C01812=1036.838,375.996,367.337,173.070,44.900,158.843
C01813=1036.829,375.750,367.377,173.063,44.896,158.841
C01814=1036.821,375.503,367.418,173.055,44.893,158.839
C01815=1036.813,375.256,367.459,173.047,44.889,158.838
C01816=1036.805,375.010,367.499,173.040,44.886,158.836
C01817=1036.796,374.763,367.540,173.033,44.883,158.835
C01818=1036.787,374.517,367.580,173.026,44.879,158.833
C01819=1036.779,374.270,367.621,173.019,44.876,158.832
C01820=1036.771,374.024,367.662,173.012,44.872,158.830
C01821=1036.763,373.778,367.703,173.005,44.869,158.828
C01822=1036.753,373.531,367.743,172.998,44.865,158.827
C01823=1036.746,373.284,367.783,172.991,44.862,158.825
C01824=1036.738,373.038,367.824,172.984,44.858,158.824
C01825=1036.729,372.791,367.865,172.976,44.855,158.822
C01826=1036.721,372.545,367.905,172.969,44.851,158.821
C01827=1036.712,372.298,367.944,172.962,44.848,158.819
C01828=1036.704,372.052,367.985,172.955,44.845,158.818
C01829=1036.696,371.805,368.026,172.948,44.841,158.816
C01830=1036.688,371.558,368.067,172.941,44.838,158.815
C01831=1036.679,371.312,368.106,172.934,44.835,158.813
C01832=1036.671,371.066,368.147,172.927,44.832,158.812
C01833=1036.664,370.819,368.187,172.921,44.828,158.810
C01834=1036.655,370.572,368.228,172.914,44.825,158.809
C01835=1036.647,370.325,368.267,172.907,44.821,158.807
C01836=1036.639,370.079,368.308,172.900,44.818,158.806
C01837=1036.631,369.832,368.348,172.893,44.814,158.804
C01838=1036.622,369.586,368.388,172.886,44.811,158.803
C01839=1036.614,369.339,368.427,172.879,44.808,158.801
C01840=1036.605,369.092,368.467,172.872,44.805,158.800
C01841=1036.596,368.846,368.507,172.865,44.802,158.798
C01842=1036.589,368.599,368.547,172.859,44.799,158.797
C01843=1036.580,368.352,368.586,172.852,44.796,158.795
C01844=1036.573,368.105,368.626,172.845,44.792,158.794
C01845=1036.564,367.859,368.666,172.838,44.789,158.792
C01846=1036.556,367.612,368.706,172.831,44.786,158.791
C01847=1036.548,367.366,368.746,172.825,44.783,158.790
C01848=1036.539,367.119,368.785,172.818,44.780,158.788
C01849=1036.531,366.872,368.825,172.811,44.777,158.787
C01850=1036.523,366.626,368.864,172.805,44.774,158.785
C01851=1036.515,366.379,368.904,172.798,44.771,158.784
C01852=1036.507,366.132,368.943,172.791,44.768,158.782
C01853=1036.499,365.885,368.983,172.785,44.764,158.781
C01854=1036.491,365.639,369.023,172.778,44.761,158.780
C01855=1036.482,365.392,369.062,172.771,44.758,158.778
C01856=1036.474,365.145,369.102,172.765,44.755,158.777
C01857=1036.466,364.899,369.141,172.758,44.752,158.775
C01858=1036.459,364.651,369.180,172.752,44.749,158.774
C01859=1036.450,364.404,369.220,172.745,44.746,158.773
C01860=1036.438,364.022,369.281,172.734,44.741,158.770
C01861=1036.426,363.640,369.342,172.725,44.737,158.768
C01862=1036.413,363.258,369.402,172.715,44.732,158.766
C01863=1036.401,362.876,369.463,172.704,44.728,158.764
C01864=1036.393,362.629,369.503,172.698,44.724,158.763
C01865=1036.385,362.382,369.542,172.692,44.721,158.761
C01866=1036.377,362.136,369.581,172.685,44.719,158.760
C01867=1036.369,361.889,369.621,172.679,44.716,158.759
C01868=1036.361,361.642,369.659,172.672,44.712,158.757
C01869=1036.353,361.395,369.699,172.666,44.710,158.756
C01870=1036.345,361.148,369.737,172.659,44.707,158.755
C01871=1036.338,360.901,369.776,172.653,44.704,158.754
C01872=1036.329,360.654,369.815,172.647,44.701,158.752
C01873=1036.321,360.407,369.854,172.640,44.699,158.751
C01874=1036.313,360.161,369.893,172.634,44.695,158.750
C01875=1036.305,359.914,369.931,172.628,44.693,158.748
C01876=1036.297,359.667,369.970,172.621,44.691,158.747
C01877=1036.289,359.420,370.008,172.615,44.687,158.746
C01878=1036.281,359.174,370.048,172.609,44.685,158.745
C01879=1036.274,358.926,370.087,172.603,44.681,158.743
C01880=1036.266,358.680,370.125,172.596,44.679,158.742
C01881=1036.258,358.432,370.164,172.590,44.676,158.741
C01882=1036.250,358.185,370.202,172.584,44.674,158.740
C01883=1036.242,357.939,370.241,172.577,44.671,158.738
C01884=1036.234,357.691,370.279,172.571,44.668,158.737
C01885=1036.226,357.446,370.318,172.565,44.666,158.736
C01886=1036.218,357.198,370.357,172.559,44.663,158.734
C01887=1036.210,356.952,370.395,172.553,44.660,158.733
C01888=1036.202,356.705,370.434,172.546,44.657,158.732
C01889=1036.195,356.458,370.472,172.541,44.655,158.731
C01890=1036.187,356.211,370.510,172.534,44.652,158.729
C01891=1036.179,355.964,370.548,172.529,44.649,158.728
C01892=1036.171,355.717,370.587,172.522,44.647,158.727
C01893=1036.163,355.469,370.625,172.516,44.644,158.726
C01894=1036.155,355.223,370.663,172.510,44.642,158.725
C01895=1036.147,354.976,370.702,172.504,44.639,158.723
C01896=1036.140,354.728,370.740,172.498,44.636,158.722
C01897=1036.132,354.482,370.777,172.491,44.634,158.721
C01898=1036.124,354.235,370.816,172.486,44.631,158.720
C01899=1036.116,353.989,370.854,172.479,44.629,158.719
C01900=1036.108,353.741,370.892,172.474,44.626,158.717
C01901=1036.101,353.494,370.930,172.467,44.624,158.716
C01902=1036.093,353.246,370.968,172.462,44.621,158.715
C01903=1036.085,353.000,371.006,172.455,44.618,158.714
C01904=1036.077,352.754,371.044,172.450,44.616,158.713
C01905=1036.069,352.506,371.082,172.443,44.614,158.711
C01906=1036.062,352.259,371.120,172.438,44.611,158.710
C01907=1036.054,352.012,371.158,172.432,44.608,158.709
C01908=1036.046,351.765,371.196,172.426,44.606,158.708
C01909=1036.039,351.518,371.234,172.420,44.604,158.707
C01910=1036.031,351.271,371.272,172.414,44.601,158.706
C01911=1036.023,351.024,371.309,172.408,44.598,158.704
C01912=1036.015,350.777,371.348,172.402,44.596,158.703
C01913=1036.008,350.530,371.385,172.396,44.594,158.702
C01914=1036.001,350.283,371.423,172.391,44.591,158.701
C01915=1035.993,350.036,371.461,172.385,44.589,158.700
C01916=1035.981,349.660,371.518,172.376,44.585,158.698
C01917=1035.969,349.284,371.575,172.367,44.581,158.696
C01918=1035.957,348.907,371.632,172.358,44.578,158.695
C01919=1035.946,348.531,371.689,172.350,44.574,158.693
C01920=1035.938,348.284,371.727,172.343,44.572,158.692
C01921=1035.931,348.037,371.765,172.338,44.570,158.691
C01922=1035.923,347.790,371.802,172.333,44.567,158.690
C01923=1035.916,347.543,371.839,172.326,44.565,158.689
C01924=1035.908,347.296,371.876,172.321,44.563,158.688
C01925=1035.900,347.048,371.914,172.315,44.560,158.686
C01926=1035.893,346.801,371.952,172.309,44.558,158.685
C01927=1035.885,346.554,371.989,172.304,44.556,158.684
C01928=1035.877,346.307,372.026,172.298,44.553,158.683
C01929=1035.869,346.060,372.063,172.292,44.551,158.682
C01930=1035.862,345.813,372.101,172.287,44.549,158.681
C01931=1035.854,345.566,372.137,172.281,44.547,158.680
C01932=1035.847,345.319,372.174,172.275,44.545,158.679
C01933=1035.840,345.072,372.212,172.270,44.542,158.678
C01934=1035.832,344.825,372.249,172.264,44.540,158.677
C01935=1035.825,344.578,372.286,172.259,44.538,158.676
C01936=1035.817,344.330,372.323,172.253,44.536,158.675
C01937=1035.810,344.083,372.360,172.247,44.533,158.674
C01938=1035.802,343.836,372.397,172.242,44.531,158.673
C01939=1035.795,343.589,372.434,172.237,44.529,158.672
C01940=1035.787,343.342,372.471,172.230,44.527,158.671
C01941=1035.780,343.094,372.508,172.225,44.525,158.670
C01942=1035.772,342.848,372.545,172.220,44.522,158.668
C01943=1035.764,342.600,372.581,172.214,44.520,158.667
C01944=1035.757,342.353,372.619,172.208,44.518,158.666
C01945=1035.749,342.106,372.655,172.203,44.516,158.665
C01946=1035.742,341.858,372.693,172.197,44.514,158.664
C01947=1035.734,341.611,372.729,172.192,44.512,158.663
C01948=1035.727,341.364,372.766,172.187,44.510,158.662
C01949=1035.719,341.116,372.803,172.181,44.508,158.661
C01950=1035.712,340.870,372.839,172.175,44.506,158.660
C01951=1035.705,340.623,372.876,172.170,44.503,158.659
C01952=1035.697,340.376,372.913,172.165,44.502,158.658
C01953=1035.689,340.128,372.949,172.160,44.500,158.657
C01954=1035.682,339.881,372.985,172.153,44.498,158.656
C01955=1035.674,339.634,373.023,172.148,44.496,158.655
C01956=1035.667,339.386,373.059,172.143,44.493,158.654
C01957=1035.660,339.140,373.095,172.138,44.492,158.653
C01958=1035.652,338.892,373.131,172.133,44.490,158.652
C01959=1035.644,338.645,373.168,172.127,44.488,158.651
C01960=1035.637,338.397,373.205,172.121,44.486,158.650
C01961=1035.629,338.150,373.241,172.116,44.483,158.649
C01962=1035.622,337.903,373.277,172.111,44.482,158.649
C01963=1035.615,337.656,373.313,172.106,44.480,158.647
C01964=1035.608,337.408,373.350,172.100,44.477,158.646
C01965=1035.600,337.161,373.386,172.095,44.476,158.646
C01966=1035.593,336.915,373.423,172.090,44.474,158.645
C01967=1035.585,336.667,373.459,172.085,44.472,158.644
C01968=1035.577,336.420,373.495,172.080,44.470,158.643
C01969=1035.570,336.172,373.532,172.073,44.468,158.642
C01970=1035.563,335.925,373.568,172.068,44.466,158.641
C01971=1035.556,335.678,373.604,172.063,44.464,158.640
C01972=1035.545,335.298,373.660,172.055,44.461,158.638
C01973=1035.533,334.919,373.715,172.048,44.458,158.637
C01974=1035.522,334.538,373.770,172.040,44.455,158.636
C01975=1035.511,334.159,373.825,172.031,44.453,158.634
C01976=1035.503,333.911,373.862,172.026,44.451,158.633
C01977=1035.496,333.665,373.897,172.021,44.449,158.632
C01978=1035.489,333.417,373.933,172.016,44.447,158.631
C01979=1035.481,333.170,373.969,172.010,44.445,158.630
C01980=1035.474,332.922,374.005,172.005,44.444,158.630
C01981=1035.466,332.675,374.041,172.000,44.442,158.629
C01982=1035.459,332.428,374.076,171.995,44.440,158.628
C01983=1035.451,332.180,374.112,171.990,44.438,158.627
C01984=1035.444,331.934,374.148,171.985,44.437,158.626
C01985=1035.437,331.686,374.183,171.980,44.435,158.625
C01986=1035.429,331.439,374.219,171.975,44.433,158.624
C01987=1035.422,331.191,374.255,171.970,44.431,158.623
C01988=1035.415,330.944,374.290,171.964,44.429,158.622
C01989=1035.408,330.696,374.326,171.959,44.428,158.622
C01990=1035.401,330.449,374.362,171.954,44.426,158.621
C01991=1035.393,330.202,374.398,171.949,44.424,158.620
C01992=1035.386,329.955,374.433,171.944,44.423,158.619
C01993=1035.379,329.706,374.469,171.939,44.421,158.618
C01994=1035.372,329.460,374.505,171.934,44.419,158.617
C01995=1035.364,329.212,374.540,171.929,44.418,158.616
C01996=1035.357,328.965,374.576,171.924,44.416,158.616
C01997=1035.350,328.718,374.611,171.919,44.414,158.615
C01998=1035.342,328.470,374.647,171.914,44.412,158.614
C01999=1035.335,328.223,374.682,171.909,44.411,158.613
C02000=1035.328,327.975,374.717,171.904,44.409,158.612
C02001=1035.320,327.728,374.752,171.899,44.407,158.611
C02002=1035.313,327.480,374.787,171.894,44.406,158.610
C02003=1035.305,327.233,374.823,171.890,44.404,158.610
C02004=1035.298,326.986,374.858,171.885,44.403,158.609
C02005=1035.290,326.738,374.893,171.880,44.401,158.608
C02006=1035.284,326.491,374.928,171.875,44.400,158.607
C02007=1035.275,326.243,374.963,171.870,44.398,158.606
C02008=1035.269,325.996,374.998,171.865,44.397,158.606
C02009=1035.261,325.749,375.032,171.860,44.395,158.605
C02010=1035.254,325.501,375.068,171.855,44.394,158.604
C02011=1035.246,325.254,375.102,171.850,44.392,158.603
C02012=1035.240,325.006,375.138,171.845,44.390,158.602
C02013=1035.231,324.758,375.172,171.840,44.389,158.602
C02014=1035.225,324.511,375.208,171.835,44.388,158.601
C02015=1035.217,324.264,375.242,171.830,44.386,158.600
C02016=1035.210,324.016,375.278,171.826,44.384,158.599
C02017=1035.202,323.769,375.312,171.821,44.383,158.598
C02018=1035.196,323.522,375.347,171.816,44.382,158.598
C02019=1035.188,323.275,375.382,171.811,44.380,158.597
C02020=1035.181,323.026,375.417,171.806,44.379,158.596
C02021=1035.173,322.779,375.452,171.801,44.377,158.595
C02022=1035.167,322.531,375.486,171.796,44.376,158.594
C02023=1035.159,322.284,375.521,171.791,44.374,158.594
C02024=1035.152,322.036,375.556,171.787,44.373,158.593
C02025=1035.144,321.789,375.591,171.783,44.372,158.592
C02026=1035.138,321.542,375.626,171.778,44.370,158.591
C02027=1035.130,321.294,375.660,171.773,44.368,158.590
C02028=1035.119,320.910,375.714,171.765,44.366,158.589
C02029=1035.108,320.526,375.768,171.758,44.364,158.588
C02030=1035.096,320.142,375.822,171.750,44.362,158.587
C02031=1035.085,319.757,375.875,171.743,44.360,158.586
C02032=1035.079,319.510,375.910,171.739,44.358,158.585
C02033=1035.071,319.262,375.944,171.734,44.357,158.584
C02034=1035.065,319.015,375.979,171.729,44.356,158.584
C02035=1035.057,318.767,376.013,171.724,44.354,158.583
C02036=1035.051,318.519,376.048,171.720,44.353,158.582
C02037=1035.043,318.272,376.082,171.715,44.351,158.581
C02038=1035.037,318.024,376.117,171.711,44.350,158.581
C02039=1035.029,317.777,376.151,171.706,44.349,158.580
C02040=1035.022,317.530,376.186,171.701,44.347,158.579
C02041=1035.015,317.282,376.220,171.697,44.346,158.578
C02042=1035.008,317.035,376.254,171.692,44.344,158.577
C02043=1035.001,316.787,376.289,171.687,44.343,158.577
C02044=1034.994,316.540,376.323,171.683,44.342,158.576
C02045=1034.987,316.292,376.358,171.678,44.340,158.575
C02046=1034.980,316.045,376.392,171.673,44.339,158.575
C02047=1034.973,315.798,376.427,171.668,44.338,158.574
C02048=1034.966,315.550,376.461,171.665,44.337,158.573
C02049=1034.959,315.302,376.495,171.660,44.335,158.572
C02050=1034.952,315.055,376.530,171.655,44.334,158.572
C02051=1034.945,314.808,376.563,171.651,44.332,158.571
C02052=1034.939,314.560,376.598,171.646,44.331,158.570
C02053=1034.932,314.313,376.632,171.641,44.330,158.570
C02054=1034.924,314.065,376.666,171.637,44.328,158.569
C02055=1034.918,313.817,376.701,171.633,44.327,158.568
C02056=1034.911,313.569,376.734,171.628,44.326,158.567
C02057=1034.904,313.322,376.770,171.624,44.325,158.567
C02058=1034.897,313.075,376.803,171.619,44.324,158.566
C02059=1034.890,312.827,376.837,171.614,44.322,158.565
C02060=1034.884,312.579,376.871,171.610,44.321,158.565
C02061=1034.876,312.331,376.905,171.606,44.320,158.564
C02062=1034.870,312.084,376.940,171.601,44.318,158.563
C02063=1034.863,311.837,376.974,171.597,44.317,158.562
C02064=1034.856,311.589,377.008,171.592,44.316,158.562
C02065=1034.849,311.342,377.041,171.587,44.315,158.561
C02066=1034.841,311.094,377.075,171.584,44.314,158.560
C02067=1034.834,310.846,377.109,171.579,44.313,158.560
C02068=1034.828,310.599,377.142,171.574,44.312,158.559
C02069=1034.820,310.352,377.175,171.570,44.310,158.558
C02070=1034.813,310.104,377.209,171.565,44.309,158.558
C02071=1034.806,309.856,377.243,171.561,44.308,158.557
C02072=1034.798,309.608,377.276,171.557,44.307,158.557
C02073=1034.791,309.361,377.310,171.552,44.306,158.556
C02074=1034.784,309.114,377.342,171.547,44.305,158.555
C02075=1034.777,308.866,377.376,171.544,44.304,158.555
C02076=1034.770,308.618,377.410,171.539,44.303,158.554
C02077=1034.763,308.371,377.444,171.534,44.302,158.553
C02078=1034.756,308.123,377.477,171.530,44.301,158.553
C02079=1034.748,307.876,377.510,171.526,44.300,158.552
C02080=1034.741,307.628,377.544,171.521,44.299,158.551
C02081=1034.734,307.380,377.577,171.517,44.297,158.551
C02082=1034.728,307.133,377.610,171.512,44.296,158.550
C02083=1034.720,306.885,377.643,171.508,44.295,158.549
C02084=1034.710,306.505,377.694,171.502,44.294,158.548
C02085=1034.698,306.126,377.746,171.494,44.292,158.547
C02086=1034.688,305.746,377.797,171.488,44.291,158.547
C02087=1034.677,305.367,377.848,171.481,44.290,158.546
C02088=1034.670,305.120,377.881,171.477,44.288,158.545
C02089=1034.663,304.872,377.914,171.473,44.287,158.544
C02090=1034.656,304.624,377.947,171.469,44.286,158.544
C02091=1034.649,304.377,377.980,171.464,44.285,158.543
C02092=1034.642,304.129,378.013,171.460,44.284,158.542
C02093=1034.636,303.881,378.046,171.456,44.283,158.542
C02094=1034.628,303.634,378.079,171.451,44.282,158.541
C02095=1034.621,303.386,378.113,171.447,44.281,158.541
C02096=1034.614,303.139,378.146,171.443,44.280,158.540
C02097=1034.607,302.890,378.179,171.439,44.280,158.539
C02098=1034.601,302.643,378.213,171.434,44.279,158.539
C02099=1034.593,302.395,378.245,171.431,44.277,158.538
C02100=1034.587,302.148,378.278,171.426,44.276,158.538
C02101=1034.580,301.900,378.312,171.422,44.276,158.537
C02102=1034.573,301.653,378.344,171.418,44.275,158.536
C02103=1034.566,301.405,378.377,171.414,44.273,158.536
C02104=1034.559,301.158,378.410,171.409,44.272,158.535
C02105=1034.552,300.909,378.443,171.406,44.272,158.535
C02106=1034.546,300.662,378.476,171.401,44.271,158.534
C02107=1034.538,300.414,378.509,171.397,44.270,158.533
C02108=1034.532,300.167,378.542,171.393,44.269,158.533
C02109=1034.525,299.919,378.575,171.389,44.268,158.532
C02110=1034.519,299.671,378.608,171.384,44.267,158.532
C02111=1034.511,299.423,378.641,171.380,44.266,158.531
C02112=1034.505,299.175,378.673,171.376,44.265,158.530
C02113=1034.498,298.928,378.706,171.372,44.264,158.530
C02114=1034.490,298.680,378.739,171.367,44.264,158.529
C02115=1034.484,298.433,378.772,171.364,44.262,158.529
C02116=1034.477,298.184,378.805,171.359,44.261,158.528
C02117=1034.471,297.937,378.838,171.355,44.261,158.528
C02118=1034.464,297.690,378.870,171.352,44.260,158.527
C02119=1034.457,297.441,378.903,171.347,44.259,158.526
C02120=1034.451,297.194,378.936,171.343,44.258,158.526
C02121=1034.444,296.946,378.969,171.339,44.257,158.525
C02122=1034.437,296.698,379.001,171.335,44.256,158.525
C02123=1034.431,296.451,379.034,171.330,44.255,158.524
C02124=1034.424,296.203,379.067,171.327,44.255,158.524
C02125=1034.417,295.955,379.099,171.323,44.253,158.523
C02126=1034.410,295.707,379.132,171.318,44.252,158.522
C02127=1034.404,295.460,379.165,171.315,44.252,158.522
C02128=1034.397,295.211,379.198,171.310,44.251,158.521
C02129=1034.390,294.964,379.230,171.307,44.250,158.521
C02130=1034.384,294.717,379.263,171.303,44.249,158.520
C02131=1034.376,294.469,379.295,171.298,44.248,158.520
C02132=1034.370,294.221,379.328,171.295,44.248,158.519
C02133=1034.363,293.973,379.359,171.290,44.247,158.518
C02134=1034.356,293.726,379.391,171.286,44.246,158.518
C02135=1034.349,293.478,379.425,171.283,44.246,158.518
C02136=1034.343,293.230,379.456,171.278,44.245,158.517
C02137=1034.336,292.982,379.489,171.275,44.244,158.516
C02138=1034.329,292.734,379.521,171.270,44.243,158.516
C02139=1034.322,292.487,379.553,171.266,44.242,158.515
C02140=1034.312,292.124,379.600,171.261,44.241,158.515
C02141=1034.301,291.761,379.647,171.255,44.241,158.514
C02142=1034.292,291.399,379.694,171.249,44.239,158.513
C02143=1034.282,291.036,379.741,171.243,44.238,158.512
C02144=1034.275,290.789,379.773,171.240,44.238,158.512
C02145=1034.268,290.540,379.805,171.235,44.237,158.511
C02146=1034.261,290.293,379.837,171.231,44.236,158.511
C02147=1034.254,290.045,379.870,171.228,44.235,158.510
C02148=1034.248,289.797,379.902,171.223,44.235,158.510
C02149=1034.241,289.549,379.933,171.220,44.234,158.509
C02150=1034.234,289.301,379.966,171.216,44.233,158.509
C02151=1034.227,289.053,379.997,171.212,44.233,158.508
C02152=1034.220,288.806,380.029,171.208,44.232,158.508
C02153=1034.214,288.558,380.061,171.205,44.231,158.507
C02154=1034.207,288.311,380.093,171.200,44.231,158.507
C02155=1034.200,288.063,380.125,171.196,44.230,158.506
C02156=1034.193,287.814,380.157,171.193,44.229,158.506
C02157=1034.186,287.567,380.189,171.188,44.229,158.505
C02158=1034.180,287.319,380.221,171.185,44.228,158.505
C02159=1034.173,287.071,380.252,171.181,44.228,158.504
C02160=1034.166,286.823,380.284,171.177,44.227,158.504
C02161=1034.159,286.576,380.316,171.173,44.226,158.503
C02162=1034.153,286.328,380.347,171.170,44.226,158.503
C02163=1034.145,286.079,380.379,171.165,44.225,158.502
C02164=1034.138,285.832,380.411,171.162,44.225,158.502
C02165=1034.132,285.584,380.443,171.158,44.224,158.501
C02166=1034.125,285.336,380.474,171.154,44.224,158.501
C02167=1034.118,285.088,380.505,171.150,44.223,158.500
C02168=1034.111,284.840,380.537,171.147,44.223,158.500
C02169=1034.105,284.592,380.568,171.142,44.222,158.500
C02170=1034.098,284.344,380.600,171.139,44.221,158.499
C02171=1034.091,284.096,380.631,171.135,44.221,158.499
C02172=1034.084,283.848,380.663,171.131,44.220,158.498
C02173=1034.077,283.601,380.695,171.127,44.220,158.498
C02174=1034.070,283.353,380.726,171.123,44.219,158.497
C02175=1034.063,283.105,380.758,171.120,44.219,158.497
C02176=1034.057,282.857,380.789,171.115,44.218,158.496
C02177=1034.049,282.609,380.820,171.112,44.217,158.496
C02178=1034.043,282.361,380.852,171.108,44.217,158.495
C02179=1034.036,282.113,380.883,171.104,44.216,158.495
C02180=1034.029,281.866,380.914,171.100,44.216,158.494
C02181=1034.022,281.618,380.946,171.097,44.215,158.494
C02182=1034.016,281.369,380.977,171.093,44.215,158.493
C02183=1034.009,281.121,381.008,171.089,44.215,158.493
C02184=1034.002,280.873,381.039,171.086,44.214,158.493
C02185=1033.996,280.625,381.071,171.082,44.213,158.492
C02186=1033.989,280.378,381.102,171.079,44.213,158.492
C02187=1033.982,280.130,381.134,171.075,44.212,158.491
C02188=1033.976,279.882,381.165,171.071,44.212,158.491
C02189=1033.969,279.634,381.197,171.067,44.211,158.490
C02190=1033.962,279.386,381.228,171.064,44.211,158.490
C02191=1033.956,279.138,381.258,171.060,44.211,158.490
C02192=1033.950,278.890,381.290,171.056,44.210,158.489
C02193=1033.943,278.642,381.321,171.052,44.209,158.489
C02194=1033.935,278.395,381.352,171.049,44.209,158.488
C02195=1033.929,278.147,381.384,171.045,44.208,158.488
C02196=1033.920,277.796,381.427,171.040,44.208,158.487
C02197=1033.910,277.445,381.471,171.035,44.207,158.486
C02198=1033.900,277.095,381.515,171.029,44.207,158.486
C02199=1033.891,276.744,381.559,171.025,44.206,158.485
C02200=1033.883,276.497,381.590,171.020,44.206,158.485
C02201=1033.877,276.248,381.620,171.017,44.205,158.484
C02202=1033.870,276.000,381.652,171.013,44.205,158.484
C02203=1033.864,275.752,381.682,171.010,44.205,158.484
C02204=1033.856,275.504,381.713,171.007,44.204,158.483
C02205=1033.850,275.256,381.744,171.002,44.204,158.483
C02206=1033.844,275.009,381.775,170.999,44.204,158.482
C02207=1033.836,274.761,381.806,170.995,44.203,158.482
C02208=1033.830,274.513,381.837,170.992,44.202,158.482
C02209=1033.823,274.265,381.868,170.988,44.202,158.481
C02210=1033.816,274.016,381.898,170.985,44.202,158.481
C02211=1033.809,273.768,381.930,170.980,44.201,158.480
C02212=1033.804,273.521,381.960,170.977,44.201,158.480
C02213=1033.796,273.272,381.990,170.974,44.201,158.480
C02214=1033.790,273.025,382.021,170.970,44.200,158.479
C02215=1033.782,272.776,382.052,170.967,44.200,158.479
C02216=1033.776,272.528,382.083,170.963,44.199,158.478
C02217=1033.770,272.281,382.113,170.959,44.199,158.478
C02218=1033.763,272.032,382.144,170.956,44.199,158.478
C02219=1033.756,271.784,382.175,170.952,44.199,158.477
C02220=1033.749,271.536,382.205,170.949,44.198,158.477
C02221=1033.742,271.288,382.236,170.945,44.198,158.476
C02222=1033.736,271.041,382.266,170.942,44.197,158.476
C02223=1033.729,270.792,382.297,170.939,44.197,158.476
C02224=1033.722,270.544,382.327,170.934,44.197,158.475
C02225=1033.716,270.296,382.358,170.931,44.196,158.475
C02226=1033.709,270.049,382.388,170.927,44.196,158.474
C02227=1033.702,269.800,382.419,170.924,44.196,158.474
C02228=1033.695,269.552,382.449,170.921,44.196,158.474
C02229=1033.689,269.303,382.480,170.917,44.195,158.473
C02230=1033.682,269.056,382.510,170.914,44.195,158.473
C02231=1033.675,268.808,382.541,170.910,44.194,158.472
C02232=1033.668,268.560,382.571,170.906,44.195,158.472
C02233=1033.662,268.312,382.601,170.903,44.194,158.472
C02234=1033.655,268.064,382.632,170.899,44.194,158.471
C02235=1033.648,267.816,382.662,170.896,44.194,158.471
C02236=1033.642,267.567,382.692,170.893,44.193,158.471
C02237=1033.635,267.320,382.722,170.889,44.193,158.470
C02238=1033.628,267.071,382.752,170.886,44.193,158.470
C02239=1033.622,266.823,382.783,170.883,44.193,158.470
C02240=1033.615,266.575,382.813,170.879,44.192,158.469
C02241=1033.608,266.327,382.843,170.876,44.192,158.469
C02242=1033.602,266.079,382.874,170.871,44.192,158.468
C02243=1033.595,265.831,382.903,170.868,44.192,158.468
C02244=1033.588,265.583,382.934,170.865,44.192,158.468
C02245=1033.581,265.335,382.964,170.861,44.192,158.467
C02246=1033.575,265.087,382.994,170.858,44.191,158.467
C02247=1033.568,264.839,383.024,170.855,44.191,158.467
C02248=1033.561,264.591,383.054,170.851,44.191,158.466
C02249=1033.555,264.343,383.085,170.848,44.190,158.466
C02250=1033.548,264.094,383.115,170.845,44.190,158.466
C02251=1033.541,263.847,383.144,170.841,44.190,158.465
C02252=1033.532,263.501,383.186,170.836,44.190,158.465
C02253=1033.522,263.155,383.227,170.831,44.190,158.464
C02254=1033.513,262.808,383.270,170.827,44.189,158.464
C02255=1033.504,262.463,383.312,170.822,44.189,158.463
C02256=1033.497,262.215,383.341,170.819,44.189,158.463
C02257=1033.490,261.966,383.371,170.816,44.189,158.463
C02258=1033.484,261.719,383.402,170.812,44.189,158.462
C02259=1033.477,261.470,383.432,170.809,44.188,158.462
C02260=1033.471,261.222,383.461,170.806,44.188,158.462
C02261=1033.464,260.974,383.491,170.801,44.188,158.461
C02262=1033.457,260.726,383.521,170.798,44.188,158.461
C02263=1033.450,260.478,383.549,170.795,44.188,158.461
C02264=1033.442,260.230,383.580,170.792,44.188,158.460
C02265=1033.436,259.982,383.609,170.788,44.188,158.460
C02266=1033.429,259.734,383.639,170.785,44.187,158.460
C02267=1033.422,259.486,383.669,170.781,44.187,158.459
C02268=1033.416,259.237,383.698,170.778,44.187,158.459
C02269=1033.408,258.989,383.728,170.775,44.187,158.459
C02270=1033.401,258.741,383.757,170.772,44.187,158.458
C02271=1033.394,258.493,383.787,170.768,44.187,158.458
C02272=1033.388,258.245,383.816,170.765,44.187,158.458
C02273=1033.381,257.997,383.846,170.762,44.187,158.458
C02274=1033.375,257.748,383.875,170.759,44.187,158.457
C02275=1033.368,257.500,383.904,170.755,44.187,158.457
C02276=1033.361,257.252,383.934,170.752,44.187,158.457
C02277=1033.354,257.004,383.963,170.749,44.187,158.456
C02278=1033.347,256.756,383.993,170.745,44.187,158.456
C02279=1033.340,256.507,384.022,170.742,44.187,158.456
C02280=1033.334,256.260,384.052,170.739,44.187,158.455
C02281=1033.327,256.011,384.081,170.735,44.187,158.455
C02282=1033.321,255.763,384.110,170.732,44.187,158.455
C02283=1033.313,255.515,384.140,170.729,44.186,158.454
C02284=1033.306,255.267,384.169,170.726,44.186,158.454
C02285=1033.300,255.018,384.198,170.722,44.186,158.454
C02286=1033.293,254.770,384.228,170.719,44.186,158.453
C02287=1033.286,254.522,384.257,170.716,44.186,158.453
C02288=1033.280,254.273,384.286,170.713,44.186,158.453
C02289=1033.273,254.026,384.316,170.709,44.186,158.453
C02290=1033.266,253.777,384.345,170.706,44.186,158.452
C02291=1033.260,253.529,384.374,170.703,44.186,158.452
C02292=1033.253,253.280,384.403,170.699,44.186,158.452
C02293=1033.246,253.033,384.433,170.696,44.186,158.451
C02294=1033.240,252.785,384.462,170.693,44.186,158.451
C02295=1033.233,252.536,384.492,170.690,44.186,158.451
C02296=1033.226,252.288,384.520,170.686,44.186,158.450
C02297=1033.219,252.040,384.550,170.683,44.186,158.450
C02298=1033.213,251.792,384.579,170.680,44.186,158.450
C02299=1033.206,251.544,384.608,170.677,44.186,158.450
C02300=1033.200,251.295,384.638,170.673,44.186,158.449
C02301=1033.193,251.047,384.667,170.670,44.186,158.449
C02302=1033.186,250.799,384.695,170.668,44.186,158.449
C02303=1033.179,250.551,384.725,170.664,44.186,158.448
C02304=1033.173,250.303,384.754,170.661,44.186,158.448
C02305=1033.167,250.054,384.783,170.658,44.186,158.448
C02306=1033.160,249.806,384.813,170.655,44.186,158.448
C02307=1033.153,249.558,384.841,170.651,44.186,158.447
C02308=1033.144,249.210,384.883,170.647,44.186,158.447
C02309=1033.135,248.863,384.923,170.643,44.186,158.447
C02310=1033.126,248.515,384.964,170.638,44.186,158.446
C02311=1033.117,248.169,385.004,170.634,44.186,158.446
C02312=1033.109,247.920,385.033,170.631,44.186,158.445
C02313=1033.103,247.672,385.062,170.627,44.186,158.445
C02314=1033.097,247.424,385.091,170.624,44.186,158.445
C02315=1033.091,247.176,385.120,170.621,44.186,158.445
C02316=1033.084,246.927,385.149,170.618,44.186,158.444
C02317=1033.077,246.679,385.178,170.616,44.186,158.444
C02318=1033.070,246.431,385.207,170.612,44.186,158.444
C02319=1033.064,246.183,385.236,170.609,44.186,158.444
C02320=1033.058,245.935,385.265,170.606,44.186,158.443
C02321=1033.051,245.686,385.294,170.603,44.186,158.443
C02322=1033.044,245.438,385.323,170.599,44.186,158.443
C02323=1033.038,245.190,385.352,170.596,44.186,158.442
C02324=1033.032,244.942,385.381,170.594,44.186,158.442
C02325=1033.025,244.694,385.410,170.590,44.186,158.442
C02326=1033.018,244.445,385.439,170.587,44.186,158.441
C02327=1033.012,244.196,385.467,170.584,44.186,158.441
C02328=1033.006,243.948,385.496,170.581,44.186,158.441
C02329=1032.999,243.700,385.525,170.578,44.186,158.441
C02330=1032.992,243.452,385.554,170.574,44.186,158.440
C02331=1032.985,243.203,385.582,170.572,44.186,158.440
C02332=1032.979,242.955,385.611,170.569,44.187,158.440
C02333=1032.972,242.707,385.639,170.566,44.187,158.440
C02334=1032.966,242.459,385.668,170.563,44.187,158.439
C02335=1032.959,242.211,385.696,170.559,44.187,158.439
C02336=1032.952,241.962,385.725,170.556,44.187,158.439
C02337=1032.945,241.714,385.754,170.554,44.187,158.439
C02338=1032.939,241.465,385.782,170.551,44.187,158.438
C02339=1032.932,241.217,385.811,170.547,44.187,158.438
C02340=1032.926,240.969,385.840,170.544,44.187,158.438
C02341=1032.919,240.721,385.867,170.541,44.188,158.438
C02342=1032.913,240.473,385.896,170.538,44.188,158.437
C02343=1032.906,240.223,385.925,170.536,44.187,158.437
C02344=1032.899,239.975,385.954,170.533,44.188,158.437
C02345=1032.892,239.728,385.982,170.529,44.188,158.437
C02346=1032.886,239.479,386.010,170.526,44.188,158.436
C02347=1032.879,239.231,386.038,170.523,44.188,158.436
C02348=1032.873,238.983,386.067,170.520,44.188,158.436
C02349=1032.866,238.735,386.095,170.517,44.188,158.436
C02350=1032.859,238.486,386.123,170.514,44.189,158.436
C02351=1032.852,238.237,386.151,170.511,44.189,158.435
C02352=1032.846,237.989,386.180,170.508,44.189,158.435
C02353=1032.839,237.741,386.208,170.505,44.189,158.435
C02354=1032.832,237.493,386.236,170.502,44.189,158.435
C02355=1032.826,237.244,386.264,170.499,44.190,158.434
C02356=1032.819,236.996,386.293,170.496,44.190,158.434
C02357=1032.812,236.748,386.321,170.493,44.190,158.434
C02358=1032.806,236.499,386.348,170.490,44.190,158.434
C02359=1032.798,236.251,386.377,170.487,44.190,158.433
C02360=1032.792,236.002,386.405,170.485,44.191,158.433
C02361=1032.785,235.754,386.433,170.481,44.191,158.433
C02362=1032.778,235.506,386.462,170.478,44.191,158.433
C02363=1032.772,235.257,386.489,170.475,44.191,158.433
C02364=1032.762,234.904,386.529,170.471,44.191,158.432
C02365=1032.753,234.551,386.570,170.466,44.192,158.432
C02366=1032.743,234.198,386.609,170.462,44.192,158.432
C02367=1032.734,233.845,386.649,170.458,44.193,158.431
C02368=1032.727,233.596,386.677,170.456,44.192,158.431
C02369=1032.721,233.348,386.706,170.453,44.193,158.431
C02370=1032.714,233.099,386.733,170.450,44.193,158.431
C02371=1032.707,232.851,386.762,170.446,44.193,158.430
C02372=1032.701,232.603,386.789,170.444,44.193,158.430
C02373=1032.694,232.354,386.817,170.441,44.193,158.430
C02374=1032.688,232.106,386.845,170.438,44.194,158.430
C02375=1032.681,231.857,386.873,170.435,44.194,158.429
C02376=1032.675,231.610,386.901,170.433,44.194,158.429
C02377=1032.668,231.362,386.929,170.429,44.194,158.429
C02378=1032.662,231.113,386.957,170.426,44.195,158.429
C02379=1032.655,230.865,386.984,170.423,44.195,158.429
C02380=1032.648,230.616,387.012,170.421,44.195,158.429
C02381=1032.641,230.368,387.040,170.418,44.195,158.428
C02382=1032.635,230.119,387.068,170.415,44.196,158.428
C02383=1032.628,229.871,387.095,170.411,44.196,158.428
C02384=1032.621,229.623,387.123,170.409,44.196,158.428
C02385=1032.615,229.374,387.151,170.406,44.196,158.427
C02386=1032.608,229.126,387.179,170.403,44.197,158.427
C02387=1032.601,228.878,387.207,170.400,44.197,158.427
C02388=1032.595,228.629,387.235,170.398,44.197,158.427
C02389=1032.588,228.381,387.263,170.395,44.197,158.427
C02390=1032.582,228.132,387.291,170.392,44.198,158.426
C02391=1032.575,227.884,387.319,170.388,44.198,158.426
C02392=1032.568,227.636,387.346,170.386,44.198,158.426
C02393=1032.561,227.387,387.373,170.383,44.199,158.426
C02394=1032.555,227.138,387.400,170.380,44.199,158.426
C02395=1032.548,226.890,387.428,170.378,44.199,158.425
C02396=1032.542,226.642,387.456,170.375,44.200,158.425
C02397=1032.534,226.394,387.483,170.372,44.200,158.425
C02398=1032.528,226.145,387.510,170.369,44.200,158.425
C02399=1032.521,225.897,387.538,170.367,44.201,158.425
C02400=1032.515,225.648,387.565,170.363,44.201,158.424
C02401=1032.508,225.399,387.593,170.360,44.201,158.424
C02402=1032.501,225.151,387.620,170.357,44.202,158.424
C02403=1032.494,224.903,387.648,170.355,44.202,158.424
C02404=1032.487,224.654,387.675,170.352,44.202,158.424
C02405=1032.481,224.406,387.703,170.349,44.203,158.424
C02406=1032.475,224.158,387.730,170.347,44.203,158.423
C02407=1032.467,223.910,387.757,170.344,44.203,158.423
C02408=1032.461,223.661,387.785,170.341,44.204,158.423
C02409=1032.454,223.413,387.812,170.338,44.204,158.423
C02410=1032.448,223.164,387.839,170.335,44.204,158.423
C02411=1032.441,222.915,387.867,170.332,44.205,158.423
C02412=1032.434,222.667,387.894,170.329,44.205,158.422
C02413=1032.427,222.419,387.922,170.327,44.205,158.422
C02414=1032.421,222.170,387.949,170.324,44.206,158.422
C02415=1032.414,221.922,387.976,170.321,44.206,158.422
C02416=1032.407,221.674,388.004,170.319,44.206,158.422
C02417=1032.401,221.425,388.031,170.316,44.207,158.421
C02418=1032.395,221.177,388.058,170.312,44.207,158.421
C02419=1032.388,220.928,388.086,170.310,44.207,158.421
C02420=1032.378,220.568,388.125,170.306,44.208,158.421
C02421=1032.369,220.207,388.165,170.302,44.208,158.421
C02422=1032.359,219.846,388.204,170.298,44.209,158.420
C02423=1032.349,219.485,388.243,170.294,44.209,158.420
C02424=1032.343,219.237,388.271,170.292,44.210,158.420
C02425=1032.336,218.988,388.297,170.288,44.210,158.420
C02426=1032.329,218.740,388.325,170.285,44.211,158.420
C02427=1032.322,218.492,388.351,170.283,44.211,158.419
C02428=1032.316,218.243,388.379,170.280,44.211,158.419
C02429=1032.309,217.994,388.405,170.277,44.212,158.419
C02430=1032.302,217.746,388.433,170.275,44.212,158.419
C02431=1032.295,217.497,388.460,170.272,44.213,158.419
C02432=1032.289,217.249,388.487,170.269,44.213,158.419
C02433=1032.282,217.001,388.513,170.267,44.213,158.418
C02434=1032.275,216.752,388.541,170.264,44.214,158.418
C02435=1032.268,216.503,388.567,170.261,44.214,158.418
C02436=1032.262,216.255,388.594,170.259,44.215,158.418
C02437=1032.255,216.007,388.621,170.256,44.215,158.418
C02438=1032.248,215.758,388.648,170.253,44.215,158.418
C02439=1032.241,215.510,388.675,170.250,44.216,158.418
C02440=1032.235,215.261,388.702,170.247,44.216,158.417
C02441=1032.228,215.013,388.728,170.245,44.217,158.417
C02442=1032.221,214.764,388.756,170.242,44.217,158.417
C02443=1032.215,214.516,388.782,170.239,44.218,158.417
C02444=1032.208,214.267,388.809,170.237,44.218,158.417
C02445=1032.201,214.019,388.836,170.234,44.218,158.417
C02446=1032.195,213.771,388.863,170.232,44.219,158.416
C02447=1032.188,213.522,388.889,170.229,44.219,158.416
C02448=1032.181,213.273,388.917,170.226,44.220,158.416
C02449=1032.175,213.025,388.943,170.223,44.220,158.416
C02450=1032.169,212.776,388.970,170.220,44.220,158.416
C02451=1032.161,212.528,388.997,170.218,44.221,158.416
C02452=1032.155,212.280,389.024,170.215,44.221,158.416
C02453=1032.148,212.031,389.050,170.212,44.222,158.415
C02454=1032.142,211.782,389.077,170.210,44.222,158.415
C02455=1032.135,211.535,389.104,170.207,44.223,158.415
C02456=1032.129,211.286,389.131,170.205,44.223,158.415
C02457=1032.122,211.037,389.158,170.202,44.223,158.415
C02458=1032.115,210.789,389.184,170.199,44.224,158.415
C02459=1032.109,210.540,389.211,170.197,44.224,158.415
C02460=1032.102,210.291,389.237,170.194,44.225,158.414
C02461=1032.095,210.044,389.264,170.192,44.225,158.414
C02462=1032.088,209.794,389.291,170.189,44.226,158.414
C02463=1032.082,209.546,389.317,170.187,44.226,158.414
C02464=1032.075,209.298,389.343,170.184,44.227,158.414
C02465=1032.068,209.049,389.370,170.181,44.228,158.414
C02466=1032.062,208.801,389.396,170.178,44.227,158.413
C02467=1032.055,208.552,389.423,170.175,44.228,158.413
C02468=1032.048,208.303,389.449,170.173,44.228,158.413
C02469=1032.041,208.055,389.475,170.170,44.229,158.413
C02470=1032.035,207.806,389.502,170.167,44.230,158.413
C02471=1032.028,207.558,389.528,170.165,44.230,158.413
C02472=1032.021,207.310,389.556,170.162,44.231,158.413
C02473=1032.014,207.061,389.582,170.160,44.231,158.413
C02474=1032.008,206.813,389.609,170.157,44.232,158.412
C02475=1032.001,206.564,389.635,170.155,44.232,158.412
C02476=1031.991,206.209,389.672,170.151,44.233,158.412
C02477=1031.981,205.854,389.710,170.147,44.234,158.412
C02478=1031.972,205.500,389.747,170.144,44.234,158.412
C02479=1031.963,205.144,389.785,170.140,44.235,158.412
C02480=1031.937,204.095,389.890,169.795,44.131,158.359
C02481=1031.930,203.847,389.915,169.792,44.133,158.359
C02482=1031.924,203.597,389.940,169.789,44.134,158.359
C02483=1031.918,203.349,389.965,169.785,44.135,158.359
C02484=1031.912,203.101,389.990,169.781,44.136,158.359
C02485=1031.906,202.852,390.014,169.777,44.137,158.359
C02486=1031.900,202.603,390.040,169.774,44.139,158.359
C02487=1031.894,202.354,390.064,169.770,44.140,158.359
C02488=1031.889,202.106,390.089,169.767,44.142,158.359
C02489=1031.882,201.857,390.114,169.764,44.143,158.359
C02490=1031.876,201.608,390.139,169.760,44.144,158.358
C02491=1031.870,201.360,390.164,169.756,44.145,158.358
C02492=1031.864,201.111,390.188,169.753,44.146,158.358
C02493=1031.858,200.862,390.214,169.749,44.148,158.358
C02494=1031.852,200.613,390.238,169.745,44.149,158.358
C02495=1031.846,200.365,390.263,169.742,44.151,158.358
C02496=1031.840,200.116,390.287,169.739,44.152,158.358
C02497=1031.833,199.867,390.312,169.735,44.153,158.358
C02498=1031.827,199.618,390.337,169.731,44.155,158.358
C02499=1031.821,199.370,390.360,169.728,44.156,158.358
C02500=1031.815,199.121,390.386,169.725,44.157,158.358
C02501=1031.808,198.872,390.410,169.721,44.159,158.358
C02502=1031.802,198.623,390.434,169.717,44.160,158.358
C02503=1031.796,198.375,390.459,169.714,44.162,158.358
C02504=1031.790,198.126,390.483,169.711,44.164,158.358
C02505=1031.783,197.877,390.507,169.707,44.165,158.358
C02506=1031.778,197.629,390.532,169.704,44.166,158.358
C02507=1031.771,197.380,390.556,169.700,44.168,158.358
C02508=1031.765,197.131,390.581,169.696,44.169,158.358
C02509=1031.759,196.882,390.605,169.693,44.170,158.358
C02510=1031.753,196.634,390.630,169.690,44.172,158.358
C02511=1031.746,196.385,390.654,169.686,44.173,158.358
C02512=1031.741,196.136,390.678,169.683,44.175,158.358
C02513=1031.734,195.887,390.702,169.679,44.177,158.358
C02514=1031.729,195.639,390.727,169.676,44.178,158.358
C02515=1031.722,195.390,390.751,169.673,44.179,158.358
C02516=1031.716,195.141,390.776,169.669,44.181,158.358
C02517=1031.710,194.893,390.800,169.665,44.182,158.358
C02518=1031.704,194.643,390.824,169.662,44.183,158.358
C02519=1031.698,194.395,390.848,169.658,44.185,158.358
C02520=1031.692,194.146,390.872,169.655,44.187,158.358
C02521=1031.685,193.898,390.897,169.652,44.188,158.358
C02522=1031.680,193.649,390.921,169.648,44.190,158.358
C02523=1031.674,193.400,390.945,169.645,44.191,158.358
C02524=1031.668,193.151,390.970,169.642,44.192,158.358
C02525=1031.662,192.902,390.994,169.638,44.194,158.358
C02526=1031.656,192.654,391.018,169.635,44.195,158.358
C02527=1031.650,192.405,391.042,169.631,44.197,158.358
C02528=1031.644,192.156,391.066,169.628,44.199,158.358
C02529=1031.638,191.907,391.090,169.625,44.200,158.358
C02530=1031.632,191.659,391.115,169.621,44.201,158.358
C02531=1031.626,191.410,391.139,169.618,44.203,158.358
C02532=1031.620,191.161,391.162,169.615,44.205,158.358
C02533=1031.614,190.912,391.187,169.612,44.206,158.358
C02534=1031.608,190.664,391.211,169.608,44.207,158.358
C02535=1031.602,190.415,391.235,169.604,44.209,158.358
C02536=1031.596,190.166,391.259,169.601,44.210,158.358
C02537=1031.590,189.917,391.283,169.597,44.211,158.358
C02538=1031.584,189.669,391.307,169.595,44.213,158.358
C02539=1031.578,189.419,391.332,169.591,44.215,158.358
C02540=1031.572,189.171,391.355,169.588,44.216,158.358
C02541=1031.565,188.888,391.383,169.584,44.218,158.358
C02542=1031.558,188.604,391.411,169.581,44.220,158.358
C02543=1031.552,188.320,391.438,169.576,44.221,158.358
C02544=1031.545,188.037,391.465,169.572,44.223,158.358
C02545=1031.539,187.788,391.490,169.570,44.225,158.358
C02546=1031.533,187.539,391.513,169.566,44.226,158.358
C02547=1031.527,187.291,391.537,169.563,44.227,158.358
C02548=1031.521,187.041,391.561,169.559,44.229,158.358
C02549=1031.516,186.792,391.585,169.557,44.231,158.358
C02550=1031.509,186.543,391.609,169.553,44.232,158.358
C02551=1031.504,186.295,391.633,169.550,44.233,158.358
C02552=1031.498,186.047,391.657,169.546,44.235,158.358
C02553=1031.491,185.797,391.680,169.544,44.237,158.358
C02554=1031.486,185.548,391.705,169.540,44.238,158.358
C02555=1031.480,185.300,391.728,169.537,44.239,158.358
C02556=1031.474,185.051,391.753,169.533,44.241,158.358
C02557=1031.468,184.803,391.776,169.531,44.243,158.358
C02558=1031.463,184.553,391.800,169.527,44.244,158.358
C02559=1031.456,184.304,391.824,169.524,44.245,158.358
C02560=1031.450,184.056,391.848,169.520,44.247,158.358
C02561=1031.445,183.808,391.872,169.517,44.249,158.358
C02562=1031.439,183.558,391.895,169.515,44.250,158.358
C02563=1031.433,183.309,391.920,169.511,44.251,158.358
C02564=1031.427,183.061,391.943,169.508,44.253,158.358
C02565=1031.421,182.811,391.967,169.504,44.255,158.358
C02566=1031.415,182.563,391.990,169.502,44.256,158.358
C02567=1031.409,182.314,392.013,169.498,44.258,158.358
C02568=1031.403,182.065,392.037,169.494,44.260,158.358
C02569=1031.396,181.817,392.060,169.492,44.262,158.358
C02570=1031.391,181.568,392.082,169.488,44.264,158.358
C02571=1031.384,181.319,392.106,169.485,44.265,158.358
C02572=1031.378,181.070,392.129,169.482,44.267,158.359
C02573=1031.372,180.821,392.153,169.479,44.268,158.359
C02574=1031.366,180.572,392.176,169.475,44.270,158.359
C02575=1031.359,180.324,392.199,169.473,44.272,158.359
C02576=1031.353,180.075,392.223,169.469,44.274,158.359
C02577=1031.347,179.826,392.246,169.466,44.276,158.359
C02578=1031.341,179.577,392.269,169.462,44.277,158.359
C02579=1031.335,179.328,392.293,169.460,44.279,158.359
C02580=1031.329,179.079,392.316,169.456,44.281,158.359
C02581=1031.322,178.831,392.339,169.452,44.283,158.359
C02582=1031.316,178.582,392.362,169.450,44.284,158.359
C02583=1031.310,178.332,392.385,169.446,44.286,158.359
C02584=1031.304,178.084,392.409,169.443,44.288,158.359
C02585=1031.298,177.835,392.432,169.440,44.290,158.359
C02586=1031.291,177.586,392.454,169.437,44.291,158.359
C02587=1031.285,177.338,392.478,169.435,44.293,158.360
C02588=1031.279,177.089,392.501,169.431,44.294,158.359
C02589=1031.274,176.840,392.524,169.428,44.296,158.360
C02590=1031.267,176.590,392.547,169.425,44.298,158.360
C02591=1031.261,176.342,392.570,169.422,44.300,158.360
C02592=1031.255,176.093,392.593,169.418,44.302,158.360
C02593=1031.249,175.845,392.616,169.415,44.303,158.360
C02594=1031.243,175.595,392.639,169.412,44.305,158.360
C02595=1031.237,175.346,392.662,169.409,44.307,158.360
C02596=1031.231,175.098,392.686,169.405,44.309,158.360
C02597=1031.225,174.849,392.708,169.403,44.310,158.360
C02598=1031.219,174.600,392.731,169.399,44.313,158.360
C02599=1031.212,174.351,392.755,169.396,44.314,158.360
C02600=1031.207,174.102,392.778,169.394,44.316,158.360
C02601=1031.200,173.853,392.800,169.390,44.317,158.360
C02602=1031.194,173.605,392.824,169.387,44.319,158.360
C02603=1031.188,173.356,392.847,169.384,44.321,158.361
C02604=1031.183,173.107,392.869,169.381,44.322,158.361
C02605=1031.176,172.823,392.895,169.377,44.325,158.361
C02606=1031.169,172.539,392.922,169.374,44.327,158.361
C02607=1031.161,172.255,392.948,169.370,44.329,158.361
C02608=1031.155,171.970,392.974,169.367,44.331,158.361
C02609=1031.149,171.722,392.997,169.364,44.332,158.361
C02610=1031.143,171.473,393.020,169.360,44.334,158.361
C02611=1031.137,171.224,393.042,169.358,44.336,158.361
C02612=1031.132,170.975,393.065,169.355,44.337,158.361
C02613=1031.126,170.727,393.089,169.351,44.340,158.361
C02614=1031.119,170.477,393.112,169.349,44.341,158.361
C02615=1031.113,170.229,393.135,169.345,44.343,158.361
C02616=1031.107,169.980,393.158,169.342,44.345,158.362
C02617=1031.101,169.731,393.181,169.340,44.347,158.362
C02618=1031.095,169.482,393.203,169.336,44.348,158.362
C02619=1031.089,169.233,393.226,169.333,44.350,158.362
C02620=1031.084,168.984,393.248,169.331,44.352,158.362
C02621=1031.078,168.735,393.271,169.327,44.354,158.362
C02622=1031.072,168.486,393.293,169.324,44.355,158.362
C02623=1031.066,168.237,393.316,169.322,44.357,158.362
C02624=1031.060,167.988,393.339,169.318,44.359,158.362
C02625=1031.054,167.740,393.362,169.315,44.361,158.362
C02626=1031.049,167.491,393.385,169.313,44.362,158.362
C02627=1031.042,167.242,393.408,169.309,44.364,158.362
C02628=1031.036,166.993,393.431,169.306,44.366,158.362
C02629=1031.031,166.744,393.453,169.304,44.367,158.362
C02630=1031.025,166.495,393.476,169.300,44.369,158.363
C02631=1031.019,166.247,393.499,169.297,44.371,158.363
C02632=1031.013,165.997,393.521,169.295,44.373,158.363
C02633=1031.007,165.748,393.544,169.291,44.375,158.363
C02634=1031.002,165.499,393.567,169.288,44.377,158.363
C02635=1030.995,165.251,393.589,169.286,44.378,158.363
C02636=1030.989,165.002,393.612,169.282,44.380,158.363
C02637=1030.984,164.753,393.635,169.279,44.382,158.363
C02638=1030.978,164.504,393.657,169.277,44.383,158.363
C02639=1030.972,164.255,393.680,169.273,44.385,158.363
C02640=1030.966,164.006,393.703,169.270,44.387,158.363
C02641=1030.960,163.757,393.726,169.268,44.388,158.363
C02642=1030.955,163.508,393.749,169.265,44.390,158.364
C02643=1030.948,163.259,393.770,169.262,44.392,158.364
C02644=1030.943,163.010,393.793,169.259,44.394,158.364
C02645=1030.937,162.761,393.816,169.256,44.396,158.364
C02646=1030.931,162.513,393.838,169.253,44.398,158.364
C02647=1030.926,162.264,393.860,169.250,44.399,158.364
C02648=1030.920,162.015,393.883,169.247,44.401,158.364
C02649=1030.914,161.766,393.906,169.245,44.403,158.364
C02650=1030.908,161.517,393.928,169.241,44.404,158.364
C02651=1030.902,161.268,393.951,169.238,44.406,158.364
C02652=1030.897,161.019,393.974,169.236,44.408,158.364
C02653=1030.891,160.770,393.997,169.233,44.409,158.364
C02654=1030.885,160.521,394.018,169.229,44.412,158.364
C02655=1030.880,160.273,394.041,169.227,44.413,158.365
C02656=1030.874,160.024,394.064,169.224,44.415,158.365
C02657=1030.868,159.775,394.085,169.221,44.417,158.365
C02658=1030.862,159.526,394.108,169.218,44.419,158.365
C02659=1030.856,159.277,394.130,169.215,44.421,158.365
C02660=1030.850,159.028,394.153,169.213,44.423,158.365
C02661=1030.844,158.779,394.175,169.209,44.424,158.365
C02662=1030.837,158.530,394.197,169.206,44.426,158.365
C02663=1030.832,158.280,394.219,169.204,44.428,158.365
C02664=1030.826,158.032,394.242,169.201,44.430,158.366
C02665=1030.820,157.783,394.263,169.197,44.432,158.366
C02666=1030.814,157.534,394.284,169.195,44.434,158.366
C02667=1030.808,157.285,394.307,169.192,44.436,158.366
C02668=1030.802,157.036,394.329,169.189,44.438,158.366
C02669=1030.795,156.752,394.355,169.186,44.440,158.366
C02670=1030.788,156.466,394.380,169.183,44.442,158.366
C02671=1030.781,156.182,394.405,169.179,44.444,158.366
C02672=1030.775,155.899,394.430,169.175,44.446,158.366
C02673=1030.768,155.649,394.452,169.173,44.448,158.367
C02674=1030.763,155.400,394.474,169.170,44.450,158.367
C02675=1030.756,155.151,394.496,169.168,44.452,158.367
C02676=1030.750,154.902,394.518,169.164,44.454,158.367
C02677=1030.744,154.653,394.540,169.161,44.456,158.367
C02678=1030.739,154.405,394.562,169.159,44.458,158.367
C02679=1030.733,154.155,394.584,169.156,44.460,158.367
C02680=1030.727,153.906,394.605,169.153,44.462,158.367
C02681=1030.720,153.658,394.628,169.150,44.464,158.368
C02682=1030.715,153.408,394.650,169.148,44.466,158.368
C02683=1030.709,153.160,394.671,169.145,44.468,158.368
C02684=1030.703,152.910,394.693,169.141,44.470,158.368
C02685=1030.697,152.661,394.715,169.139,44.472,158.368
C02686=1030.690,152.413,394.737,169.136,44.474,158.368
C02687=1030.684,152.163,394.759,169.132,44.475,158.368
C02688=1030.679,151.915,394.780,169.130,44.477,158.368
C02689=1030.673,151.665,394.802,169.127,44.479,158.368
C02690=1030.667,151.416,394.824,169.125,44.481,158.369
C02691=1030.661,151.168,394.846,169.121,44.483,158.369
C02692=1030.655,150.919,394.867,169.119,44.485,158.369
C02693=1030.649,150.670,394.889,169.116,44.487,158.369
C02694=1030.643,150.421,394.911,169.113,44.489,158.369
C02695=1030.637,150.172,394.932,169.111,44.491,158.369
C02696=1030.631,149.923,394.953,169.107,44.493,158.369
C02697=1030.625,149.674,394.976,169.105,44.495,158.369
C02698=1030.619,149.425,394.998,169.102,44.497,158.370
C02699=1030.613,149.176,395.020,169.100,44.499,158.370
C02700=1030.607,148.927,395.041,169.096,44.501,158.370
C02701=1030.601,148.678,395.063,169.093,44.503,158.370
C02702=1030.595,148.429,395.084,169.091,44.505,158.370
C02703=1030.589,148.180,395.106,169.088,44.507,158.370
C02704=1030.583,147.931,395.127,169.086,44.509,158.370
C02705=1030.577,147.682,395.149,169.082,44.511,158.371
C02706=1030.571,147.433,395.170,169.080,44.513,158.371
C02707=1030.566,147.184,395.192,169.077,44.515,158.371
C02708=1030.559,146.935,395.213,169.074,44.516,158.371
C02709=1030.553,146.686,395.235,169.072,44.518,158.371
C02710=1030.547,146.437,395.257,169.068,44.521,158.371
C02711=1030.541,146.188,395.278,169.066,44.522,158.371
C02712=1030.535,145.939,395.299,169.063,44.524,158.371
C02713=1030.529,145.690,395.321,169.061,44.527,158.372
C02714=1030.524,145.441,395.342,169.057,44.529,158.372
C02715=1030.517,145.192,395.364,169.055,44.531,158.372
C02716=1030.511,144.943,395.386,169.052,44.533,158.372
C02717=1030.505,144.694,395.406,169.049,44.535,158.372
C02718=1030.499,144.445,395.427,169.047,44.537,158.372
C02719=1030.493,144.196,395.449,169.043,44.539,158.372
C02720=1030.487,143.947,395.470,169.041,44.541,158.373
C02721=1030.481,143.698,395.492,169.038,44.543,158.373
C02722=1030.475,143.449,395.513,169.036,44.545,158.373
C02723=1030.469,143.200,395.535,169.033,44.547,158.373
C02724=1030.463,142.951,395.555,169.030,44.549,158.373
C02725=1030.457,142.701,395.577,169.027,44.551,158.373
C02726=1030.451,142.453,395.598,169.025,44.553,158.374
C02727=1030.445,142.204,395.620,169.022,44.555,158.374
C02728=1030.439,141.954,395.641,169.019,44.557,158.374
C02729=1030.434,141.705,395.662,169.016,44.559,158.374
C02730=1030.427,141.456,395.683,169.013,44.561,158.374
C02731=1030.421,141.208,395.704,169.011,44.563,158.374
C02732=1030.415,140.959,395.726,169.008,44.565,158.374
C02733=1030.409,140.673,395.750,169.005,44.568,158.375
C02734=1030.402,140.389,395.774,169.002,44.570,158.375
C02735=1030.395,140.104,395.798,168.999,44.572,158.375
C02736=1030.387,139.819,395.823,168.996,44.575,158.375
C02737=1030.382,139.570,395.843,168.993,44.577,158.375
C02738=1030.376,139.321,395.865,168.990,44.579,158.375
C02739=1030.370,139.073,395.886,168.988,44.581,158.375
C02740=1030.364,138.823,395.907,168.985,44.583,158.376
C02741=1030.358,138.574,395.929,168.982,44.584,158.376
C02742=1030.352,138.325,395.949,168.980,44.586,158.376
C02743=1030.346,138.076,395.970,168.976,44.589,158.376
C02744=1030.341,137.827,395.992,168.974,44.591,158.376
C02745=1030.334,137.578,396.012,168.971,44.593,158.376
C02746=1030.328,137.329,396.033,168.969,44.595,158.377
C02747=1030.322,137.080,396.055,168.966,44.597,158.377
C02748=1030.316,136.830,396.075,168.964,44.599,158.377
C02749=1030.310,136.582,396.096,168.960,44.602,158.377
C02750=1030.304,136.332,396.117,168.958,44.604,158.377
C02751=1030.298,136.084,396.138,168.955,44.606,158.377
C02752=1030.292,135.834,396.159,168.953,44.608,158.377
C02753=1030.286,135.586,396.180,168.950,44.609,158.378
C02754=1030.280,135.336,396.201,168.948,44.612,158.378
C02755=1030.274,135.087,396.222,168.944,44.614,158.378
C02756=1030.268,134.838,396.242,168.942,44.616,158.378
C02757=1030.262,134.589,396.263,168.939,44.618,158.378
C02758=1030.256,134.340,396.284,168.936,44.620,158.378
C02759=1030.250,134.091,396.305,168.934,44.622,158.378
C02760=1030.244,133.842,396.325,168.932,44.625,158.379
C02761=1030.238,133.593,396.347,168.929,44.626,158.379
C02762=1030.232,133.344,396.367,168.926,44.628,158.379
C02763=1030.226,133.095,396.388,168.923,44.631,158.379
C02764=1030.220,132.846,396.409,168.920,44.633,158.379
C02765=1030.214,132.597,396.430,168.918,44.635,158.380
C02766=1030.208,132.348,396.451,168.915,44.637,158.380
C02767=1030.203,132.098,396.471,168.913,44.639,158.380
C02768=1030.196,131.850,396.492,168.910,44.641,158.380
C02769=1030.190,131.600,396.513,168.908,44.643,158.380
C02770=1030.183,131.351,396.534,168.905,44.645,158.380
C02771=1030.178,131.102,396.554,168.902,44.648,158.380
C02772=1030.172,130.853,396.575,168.899,44.650,158.381
C02773=1030.166,130.604,396.596,168.897,44.652,158.381
C02774=1030.160,130.356,396.616,168.894,44.653,158.381
C02775=1030.154,130.106,396.637,168.892,44.656,158.381
C02776=1030.148,129.857,396.657,168.889,44.658,158.381
C02777=1030.141,129.608,396.678,168.887,44.660,158.381
C02778=1030.135,129.359,396.698,168.883,44.663,158.382
C02779=1030.129,129.109,396.719,168.881,44.665,158.382
C02780=1030.123,128.861,396.739,168.878,44.667,158.382
C02781=1030.117,128.611,396.759,168.876,44.669,158.382
C02782=1030.111,128.363,396.780,168.873,44.671,158.382
C02783=1030.105,128.113,396.801,168.871,44.673,158.383
C02784=1030.099,127.864,396.821,168.867,44.676,158.383
C02785=1030.092,127.615,396.841,168.865,44.678,158.383
C02786=1030.086,127.366,396.861,168.862,44.680,158.383
C02787=1030.081,127.117,396.882,168.860,44.682,158.383
C02788=1030.074,126.868,396.902,168.857,44.684,158.383
C02789=1030.068,126.619,396.922,168.855,44.686,158.384
C02790=1030.061,126.370,396.943,168.852,44.689,158.384
C02791=1030.056,126.120,396.963,168.850,44.691,158.384
C02792=1030.050,125.871,396.984,168.846,44.693,158.384
C02793=1030.044,125.622,397.004,168.844,44.696,158.384
C02794=1030.038,125.373,397.024,168.841,44.698,158.384
C02795=1030.031,125.124,397.045,168.839,44.700,158.385
C02796=1030.025,124.875,397.065,168.836,44.702,158.385
C02797=1030.018,124.590,397.088,168.833,44.704,158.385
C02798=1030.012,124.305,397.111,168.830,44.707,158.385
C02799=1030.005,124.019,397.134,168.827,44.710,158.386
C02800=1029.997,123.735,397.157,168.825,44.712,158.386
C02801=1029.991,123.486,397.177,168.822,44.714,158.386
C02802=1029.986,123.236,397.198,168.820,44.716,158.386
C02803=1029.980,122.988,397.218,168.816,44.718,158.386
C02804=1029.974,122.739,397.238,168.814,44.720,158.386
C02805=1029.967,122.490,397.259,168.811,44.723,158.387
C02806=1029.961,122.241,397.280,168.809,44.725,158.387
C02807=1029.955,121.992,397.299,168.806,44.727,158.387
C02808=1029.949,121.743,397.320,168.804,44.729,158.387
C02809=1029.943,121.494,397.340,168.801,44.731,158.387
C02810=1029.937,121.245,397.360,168.799,44.733,158.387
C02811=1029.931,120.994,397.380,168.796,44.735,158.388
C02812=1029.925,120.746,397.400,168.794,44.738,158.388
C02813=1029.919,120.497,397.420,168.791,44.740,158.388
C02814=1029.913,120.247,397.440,168.789,44.742,158.388
C02815=1029.907,119.998,397.461,168.786,44.744,158.388
C02816=1029.901,119.749,397.481,168.783,44.747,158.388
C02817=1029.895,119.501,397.501,168.780,44.749,158.389
C02818=1029.889,119.251,397.521,168.778,44.751,158.389
C02819=1029.883,119.002,397.541,168.775,44.753,158.389
C02820=1029.878,118.753,397.561,168.773,44.755,158.389
C02821=1029.872,118.504,397.581,168.770,44.757,158.389
C02822=1029.865,118.255,397.602,168.768,44.759,158.389
C02823=1029.859,118.006,397.622,168.765,44.762,158.390
C02824=1029.853,117.757,397.642,168.763,44.764,158.390
C02825=1029.848,117.507,397.662,168.760,44.765,158.390
C02826=1029.841,117.258,397.682,168.758,44.767,158.390
C02827=1029.835,117.009,397.702,168.755,44.770,158.390
C02828=1029.829,116.760,397.722,168.753,44.772,158.390
C02829=1029.823,116.511,397.742,168.750,44.774,158.391
C02830=1029.818,116.262,397.763,168.748,44.776,158.391
C02831=1029.812,116.012,397.782,168.745,44.779,158.391
C02832=1029.806,115.763,397.802,168.743,44.780,158.391
C02833=1029.800,115.515,397.822,168.740,44.782,158.391
C02834=1029.794,115.266,397.842,168.737,44.784,158.391
C02835=1029.788,115.016,397.863,168.735,44.787,158.392
C02836=1029.782,114.767,397.883,168.733,44.789,158.392
C02837=1029.776,114.518,397.902,168.730,44.791,158.392
C02838=1029.770,114.269,397.922,168.727,44.793,158.392
C02839=1029.764,114.020,397.942,168.725,44.796,158.392
C02840=1029.758,113.771,397.962,168.723,44.797,158.393
C02841=1029.753,113.521,397.982,168.720,44.799,158.393
C02842=1029.747,113.272,398.002,168.717,44.801,158.393
C02843=1029.741,113.023,398.022,168.715,44.803,158.393
C02844=1029.735,112.774,398.041,168.713,44.806,158.393
C02845=1029.729,112.525,398.061,168.710,44.808,158.393
C02846=1029.723,112.275,398.081,168.708,44.811,158.394
C02847=1029.717,112.026,398.101,168.704,44.813,158.394
C02848=1029.711,111.777,398.121,168.702,44.815,158.394
C02849=1029.705,111.528,398.141,168.699,44.817,158.394
C02850=1029.699,111.279,398.160,168.697,44.819,158.394
C02851=1029.693,111.030,398.179,168.694,44.821,158.394
C02852=1029.686,110.780,398.199,168.692,44.824,158.395
C02853=1029.680,110.531,398.219,168.689,44.826,158.395
C02854=1029.674,110.283,398.239,168.687,44.828,158.395
C02855=1029.669,110.033,398.258,168.684,44.830,158.395
C02856=1029.663,109.784,398.278,168.682,44.832,158.395
C02857=1029.656,109.534,398.298,168.679,44.835,158.396
C02858=1029.650,109.286,398.317,168.677,44.837,158.396
C02859=1029.644,109.036,398.336,168.675,44.840,158.396
C02860=1029.638,108.788,398.356,168.672,44.841,158.396
C02861=1029.631,108.503,398.378,168.669,44.844,158.396
C02862=1029.624,108.217,398.400,168.666,44.847,158.397
C02863=1029.617,107.932,398.422,168.663,44.849,158.397
C02864=1029.610,107.647,398.444,168.660,44.852,158.397
C02865=1029.604,107.398,398.464,168.658,44.854,158.397
C02866=1029.598,107.149,398.484,168.656,44.856,158.397
C02867=1029.591,106.900,398.503,168.653,44.858,158.398
C02868=1029.585,106.650,398.523,168.651,44.861,158.398
C02869=1029.579,106.401,398.542,168.648,44.863,158.398
C02870=1029.574,106.152,398.562,168.646,44.866,158.398
C02871=1029.567,105.903,398.580,168.643,44.867,158.398
C02872=1029.561,105.654,398.600,168.641,44.869,158.399
C02873=1029.555,105.404,398.620,168.638,44.872,158.399
C02874=1029.549,105.156,398.639,168.636,44.874,158.399
C02875=1029.543,104.906,398.658,168.633,44.877,158.399
C02876=1029.537,104.657,398.677,168.630,44.879,158.399
C02877=1029.531,104.408,398.697,168.627,44.881,158.399
C02878=1029.525,104.159,398.716,168.625,44.883,158.400
C02879=1029.519,103.909,398.736,168.622,44.885,158.400
C02880=1029.513,103.660,398.756,168.620,44.887,158.400
C02881=1029.507,103.411,398.775,168.618,44.890,158.400
C02882=1029.500,103.162,398.794,168.615,44.892,158.400
C02883=1029.494,102.913,398.813,168.613,44.895,158.401
C02884=1029.489,102.663,398.833,168.610,44.897,158.401
C02885=1029.482,102.414,398.851,168.608,44.898,158.401
C02886=1029.476,102.165,398.871,168.605,44.901,158.401
C02887=1029.471,101.916,398.891,168.603,44.903,158.401
C02888=1029.465,101.666,398.910,168.600,44.905,158.401
C02889=1029.459,101.417,398.928,168.598,44.908,158.402
C02890=1029.453,101.169,398.948,168.595,44.910,158.402
C02891=1029.447,100.919,398.968,168.593,44.912,158.402
C02892=1029.440,100.670,398.986,168.590,44.914,158.402
C02893=1029.435,100.421,399.006,168.588,44.916,158.402
C02894=1029.429,100.172,399.026,168.585,44.919,158.403
C02895=1029.423,99.922,399.045,168.583,44.921,158.403
C02896=1029.417,99.673,399.063,168.580,44.923,158.403
C02897=1029.410,99.424,399.082,168.578,44.925,158.403
C02898=1029.405,99.175,399.101,168.575,44.927,158.403
C02899=1029.398,98.926,399.120,168.573,44.930,158.404
C02900=1029.392,98.676,399.139,168.571,44.932,158.404
C02901=1029.386,98.428,399.159,168.568,44.935,158.404
C02902=1029.380,98.178,399.178,168.566,44.937,158.404
C02903=1029.374,97.929,399.196,168.563,44.939,158.404
C02904=1029.368,97.680,399.216,168.561,44.941,158.405
C02905=1029.361,97.430,399.234,168.559,44.944,158.405
C02906=1029.355,97.181,399.253,168.556,44.946,158.405
C02907=1029.349,96.932,399.272,168.554,44.948,158.405
C02908=1029.343,96.683,399.291,168.551,44.950,158.405
C02909=1029.337,96.433,399.310,168.549,44.953,158.406
C02910=1029.331,96.184,399.329,168.546,44.955,158.406
C02911=1029.325,95.935,399.348,168.544,44.957,158.406
C02912=1029.319,95.686,399.367,168.541,44.960,158.406
C02913=1029.312,95.437,399.385,168.539,44.962,158.406
C02914=1029.307,95.187,399.405,168.536,44.964,158.407
C02915=1029.300,94.938,399.423,168.534,44.966,158.407
C02916=1029.294,94.689,399.442,168.532,44.969,158.407
C02917=1029.288,94.439,399.461,168.529,44.971,158.407
C02918=1029.282,94.190,399.480,168.527,44.973,158.407
C02919=1029.276,93.941,399.499,168.524,44.975,158.407
C02920=1029.270,93.692,399.518,168.522,44.977,158.408
C02921=1029.264,93.443,399.537,168.519,44.980,158.408
C02922=1029.258,93.194,399.555,168.517,44.982,158.408
C02923=1029.252,92.945,399.574,168.514,44.985,158.408
C02924=1029.246,92.695,399.593,168.512,44.987,158.408
C02925=1029.238,92.386,399.616,168.509,44.989,158.409
C02926=1029.231,92.078,399.640,168.506,44.992,158.409
C02927=1029.223,91.770,399.663,168.503,44.995,158.409
C02928=1029.216,91.461,399.686,168.500,44.998,158.409
C02929=1029.210,91.211,399.705,168.497,45.000,158.409
C02930=1029.204,90.962,399.724,168.495,45.002,158.410
C02931=1029.197,90.713,399.743,168.492,45.004,158.410
C02932=1029.192,90.463,399.762,168.490,45.007,158.410
C02933=1029.185,90.214,399.781,168.487,45.009,158.410
C02934=1029.180,89.965,399.799,168.485,45.011,158.410
C02935=1029.174,89.716,399.817,168.482,45.014,158.411
C02936=1029.168,89.467,399.836,168.480,45.016,158.411
C02937=1029.161,89.218,399.855,168.478,45.018,158.411
C02938=1029.155,88.968,399.873,168.475,45.020,158.411
C02939=1029.149,88.718,399.892,168.473,45.023,158.411
C02940=1029.143,88.469,399.910,168.470,45.026,158.412
C02941=1029.136,88.220,399.929,168.468,45.028,158.412
C02942=1029.130,87.970,399.947,168.465,45.030,158.412
C02943=1029.125,87.722,399.965,168.463,45.032,158.412
C02944=1029.118,87.473,399.984,168.461,45.035,158.413
C02945=1029.112,87.224,400.003,168.458,45.037,158.413
C02946=1029.106,86.974,400.021,168.456,45.039,158.413
C02947=1029.100,86.725,400.040,168.453,45.041,158.413
C02948=1029.093,86.476,400.058,168.451,45.044,158.413
C02949=1029.087,86.226,400.076,168.448,45.046,158.413
C02950=1029.081,85.977,400.095,168.446,45.049,158.414
C02951=1029.075,85.728,400.113,168.443,45.051,158.414
C02952=1029.069,85.478,400.131,168.441,45.053,158.414
C02953=1029.063,85.241,400.149,168.439,45.055,158.414
C02954=1029.057,85.004,400.166,168.436,45.058,158.415
C02955=1029.051,84.766,400.184,168.435,45.060,158.415
C02956=1029.045,84.529,400.202,168.432,45.062,158.415
C02957=1029.039,84.291,400.219,168.430,45.064,158.415
C02958=1029.034,84.054,400.236,168.427,45.066,158.415
C02959=1029.028,83.817,400.254,168.425,45.068,158.415
C02960=1029.023,83.579,400.272,168.422,45.071,158.416
C02961=1029.016,83.330,400.290,168.420,45.073,158.416
C02962=1029.010,83.080,400.308,168.418,45.076,158.416
C02963=1029.004,82.831,400.327,168.415,45.078,158.416
C02964=1028.998,82.582,400.344,168.413,45.080,158.416
C02965=1028.992,82.333,400.363,168.410,45.082,158.417
C02966=1028.986,82.083,400.381,168.408,45.085,158.417
C02967=1028.979,81.834,400.400,168.405,45.087,158.417
C02968=1028.973,81.586,400.418,168.403,45.089,158.417
C02969=1028.967,81.336,400.436,168.400,45.091,158.417
C02970=1028.962,81.087,400.455,168.399,45.093,158.418
C02971=1028.955,80.837,400.473,168.397,45.096,158.418
C02972=1028.950,80.589,400.491,168.394,45.098,158.418
C02973=1028.943,80.339,400.509,168.392,45.101,158.418
C02974=1028.937,80.090,400.528,168.389,45.102,158.418
C02975=1028.931,79.840,400.546,168.387,45.105,158.419
C02976=1028.925,79.591,400.564,168.384,45.107,158.419
C02977=1028.919,79.342,400.582,168.382,45.109,158.419
C02978=1028.913,79.093,400.601,168.379,45.112,158.419
C02979=1028.907,78.844,400.618,168.377,45.114,158.419
C02980=1028.901,78.594,400.637,168.375,45.116,158.420
C02981=1028.895,78.345,400.655,168.372,45.118,158.420
C02982=1028.888,78.096,400.674,168.370,45.121,158.420
C02983=1028.883,77.846,400.692,168.367,45.123,158.420
C02984=1028.876,77.597,400.709,168.365,45.125,158.420
C02985=1028.870,77.348,400.728,168.362,45.128,158.420
C02986=1028.865,77.099,400.745,168.360,45.130,158.421
C02987=1028.858,76.850,400.764,168.357,45.132,158.421
C02988=1028.852,76.600,400.782,168.355,45.134,158.421
C02989=1028.845,76.314,400.803,168.352,45.137,158.421
C02990=1028.838,76.030,400.823,168.349,45.140,158.421
C02991=1028.831,75.745,400.844,168.347,45.142,158.422
C02992=1028.824,75.459,400.863,168.344,45.145,158.422
C02993=1028.818,75.210,400.882,168.341,45.148,158.422
C02994=1028.812,74.961,400.900,168.339,45.150,158.422
C02995=1028.806,74.711,400.918,168.336,45.153,158.423
C02996=1028.800,74.462,400.936,168.334,45.155,158.423
C02997=1028.793,74.213,400.953,168.331,45.157,158.423
C02998=1028.787,73.963,400.971,168.329,45.159,158.423
C02999=1028.781,73.714,400.989,168.327,45.162,158.423
C03000=1028.775,73.465,401.007,168.324,45.164,158.424
C03001=1028.769,73.215,401.025,168.322,45.167,158.424
C03002=1028.763,72.967,401.042,168.319,45.169,158.424
C03003=1028.756,72.717,401.060,168.317,45.171,158.424
C03004=1028.750,72.468,401.079,168.314,45.173,158.424
C03005=1028.745,72.219,401.096,168.312,45.176,158.425
C03006=1028.738,71.969,401.114,168.309,45.178,158.425
C03007=1028.732,71.719,401.132,168.307,45.181,158.425
C03008=1028.726,71.470,401.149,168.305,45.183,158.425
C03009=1028.720,71.221,401.168,168.302,45.185,158.425
C03010=1028.714,70.972,401.185,168.300,45.187,158.425
C03011=1028.707,70.723,401.203,168.298,45.190,158.426
C03012=1028.701,70.473,401.221,168.296,45.192,158.426
C03013=1028.696,70.224,401.238,168.294,45.194,158.426
C03014=1028.689,69.974,401.256,168.291,45.196,158.426
C03015=1028.683,69.726,401.273,168.289,45.199,158.427
C03016=1028.677,69.476,401.292,168.286,45.201,158.427
C03017=1028.671,69.227,401.310,168.284,45.203,158.427
C03018=1028.665,68.978,401.327,168.281,45.206,158.427
C03019=1028.658,68.728,401.345,168.279,45.208,158.427
C03020=1028.653,68.479,401.362,168.276,45.210,158.427
C03021=1028.647,68.229,401.380,168.274,45.213,158.428
C03022=1028.640,67.980,401.398,168.272,45.215,158.428
C03023=1028.634,67.731,401.415,168.269,45.218,158.428
C03024=1028.627,67.482,401.432,168.267,45.220,158.428
C03025=1028.622,67.233,401.450,168.264,45.222,158.429
C03026=1028.616,66.983,401.468,168.262,45.224,158.429
C03027=1028.610,66.734,401.485,168.260,45.227,158.429
C03028=1028.603,66.484,401.503,168.257,45.229,158.429
C03029=1028.597,66.235,401.521,168.255,45.232,158.429
C03030=1028.591,65.986,401.538,168.252,45.234,158.429
C03031=1028.585,65.736,401.556,168.250,45.236,158.430
C03032=1028.579,65.487,401.573,168.247,45.238,158.430
C03033=1028.573,65.238,401.591,168.245,45.241,158.430
C03034=1028.566,64.989,401.608,168.242,45.243,158.430
C03035=1028.560,64.739,401.626,168.240,45.246,158.430
C03036=1028.554,64.490,401.642,168.238,45.248,158.431
C03037=1028.548,64.241,401.660,168.235,45.250,158.431
C03038=1028.542,63.992,401.678,168.233,45.252,158.431
C03039=1028.535,63.742,401.695,168.230,45.255,158.431
C03040=1028.530,63.493,401.713,168.228,45.257,158.431
C03041=1028.523,63.243,401.730,168.226,45.260,158.432
C03042=1028.517,62.994,401.746,168.223,45.262,158.432
C03043=1028.511,62.745,401.764,168.221,45.264,158.432
C03044=1028.504,62.495,401.782,168.218,45.267,158.432
C03045=1028.498,62.247,401.799,168.216,45.270,158.433
C03046=1028.491,61.996,401.815,168.213,45.272,158.433
C03047=1028.486,61.747,401.833,168.210,45.274,158.433
C03048=1028.479,61.498,401.850,168.208,45.277,158.433
C03049=1028.473,61.249,401.867,168.205,45.279,158.433
C03050=1028.467,60.999,401.884,168.203,45.282,158.434
C03051=1028.461,60.750,401.901,168.201,45.285,158.434
C03052=1028.454,60.501,401.919,168.198,45.287,158.434
C03053=1028.447,60.216,401.938,168.196,45.289,158.434
C03054=1028.440,59.930,401.958,168.193,45.292,158.434
C03055=1028.433,59.645,401.977,168.190,45.295,158.435
C03056=1028.425,59.360,401.997,168.187,45.298,158.435
C03057=1028.419,59.110,402.014,168.185,45.300,158.435
C03058=1028.412,58.861,402.031,168.182,45.303,158.435
C03059=1028.407,58.612,402.049,168.180,45.305,158.436
C03060=1028.400,58.362,402.065,168.178,45.308,158.436
C03061=1028.394,58.113,402.082,168.175,45.310,158.436
C03062=1028.387,57.864,402.099,168.173,45.312,158.436
C03063=1028.382,57.614,402.116,168.170,45.315,158.436
C03064=1028.375,57.365,402.134,168.168,45.317,158.437
C03065=1028.369,57.116,402.151,168.166,45.320,158.437
C03066=1028.362,56.866,402.167,168.163,45.322,158.437
C03067=1028.357,56.617,402.185,168.161,45.324,158.437
C03068=1028.351,56.367,402.201,168.158,45.327,158.437
C03069=1028.344,56.118,402.218,168.156,45.329,158.438
C03070=1028.338,55.869,402.235,168.154,45.332,158.438
C03071=1028.332,55.619,402.253,168.151,45.334,158.438
C03072=1028.326,55.370,402.270,168.149,45.336,158.438
C03073=1028.319,55.120,402.286,168.146,45.338,158.438
C03074=1028.313,54.871,402.303,168.144,45.341,158.439
C03075=1028.307,54.622,402.321,168.142,45.344,158.439
C03076=1028.301,54.372,402.337,168.139,45.346,158.439
C03077=1028.295,54.124,402.354,168.137,45.348,158.439
C03078=1028.288,53.874,402.371,168.134,45.350,158.439
C03079=1028.283,53.624,402.388,168.132,45.353,158.440
C03080=1028.277,53.375,402.405,168.129,45.355,158.440
C03081=1028.270,53.126,402.422,168.127,45.358,158.440
C03082=1028.264,52.876,402.438,168.124,45.360,158.440
C03083=1028.258,52.627,402.456,168.122,45.363,158.440
C03084=1028.251,52.378,402.473,168.120,45.365,158.441
C03085=1028.245,52.129,402.490,168.117,45.367,158.441
C03086=1028.239,51.880,402.506,168.115,45.370,158.441
C03087=1028.233,51.630,402.523,168.112,45.372,158.441
C03088=1028.227,51.381,402.541,168.110,45.375,158.441
C03089=1028.221,51.131,402.557,168.108,45.377,158.442
C03090=1028.215,50.881,402.574,168.105,45.379,158.442
C03091=1028.208,50.633,402.591,168.103,45.381,158.442
C03092=1028.203,50.383,402.607,168.100,45.384,158.442
C03093=1028.196,50.133,402.625,168.098,45.386,158.442
C03094=1028.190,49.884,402.641,168.096,45.389,158.443
C03095=1028.184,49.635,402.658,168.093,45.391,158.443
C03096=1028.178,49.385,402.675,168.091,45.393,158.443
C03097=1028.172,49.136,402.692,168.088,45.395,158.443
C03098=1028.166,48.887,402.708,168.086,45.397,158.443
C03099=1028.159,48.637,402.725,168.083,45.400,158.443
C03100=1028.153,48.388,402.742,168.081,45.402,158.444
C03101=1028.148,48.139,402.759,168.079,45.405,158.444
C03102=1028.142,47.890,402.776,168.076,45.407,158.444
C03103=1028.135,47.640,402.792,168.074,45.409,158.444
C03104=1028.129,47.390,402.809,168.071,45.411,158.444
C03105=1028.123,47.142,402.826,168.069,45.414,158.445
C03106=1028.118,46.892,402.843,168.066,45.416,158.445
C03107=1028.111,46.643,402.860,168.064,45.419,158.445
C03108=1028.105,46.393,402.876,168.061,45.421,158.445
C03109=1028.099,46.144,402.892,168.059,45.423,158.445
C03110=1028.093,45.895,402.909,168.057,45.426,158.445
C03111=1028.087,45.645,402.927,168.054,45.428,158.446
C03112=1028.081,45.395,402.943,168.052,45.430,158.446
C03113=1028.075,45.147,402.960,168.049,45.432,158.446
C03114=1028.069,44.897,402.976,168.047,45.434,158.446
C03115=1028.062,44.647,402.993,168.044,45.437,158.446
C03116=1028.057,44.398,403.010,168.042,45.439,158.446
C03117=1028.050,44.113,403.028,168.038,45.442,158.447
C03118=1028.042,43.827,403.048,168.036,45.445,158.447
C03119=1028.036,43.541,403.067,168.034,45.447,158.447
C03120=1028.029,43.256,403.086,168.030,45.450,158.447
C03121=1028.023,43.006,403.103,168.028,45.452,158.447
C03122=1028.017,42.757,403.119,168.025,45.454,158.448
C03123=1028.011,42.507,403.135,168.023,45.457,158.448
C03124=1028.005,42.258,403.152,168.021,45.459,158.448
C03125=1027.998,42.010,403.168,168.018,45.462,158.448
C03126=1027.992,41.760,403.185,168.016,45.464,158.448
C03127=1027.986,41.510,403.201,168.014,45.466,158.449
C03128=1027.980,41.261,403.217,168.011,45.468,158.449
C03129=1027.974,41.011,403.233,168.009,45.471,158.449
C03130=1027.968,40.762,403.250,168.006,45.473,158.449
C03131=1027.962,40.512,403.266,168.004,45.476,158.449
C03132=1027.956,40.263,403.283,168.001,45.478,158.449
C03133=1027.950,40.013,403.299,167.999,45.480,158.450
C03134=1027.943,39.765,403.316,167.996,45.482,158.450
C03135=1027.937,39.515,403.332,167.994,45.485,158.450
C03136=1027.931,39.265,403.349,167.992,45.487,158.450
C03137=1027.925,39.016,403.365,167.989,45.490,158.450
C03138=1027.918,38.767,403.381,167.987,45.492,158.451
C03139=1027.912,38.518,403.397,167.984,45.495,158.451
C03140=1027.906,38.268,403.413,167.982,45.497,158.451
C03141=1027.900,38.019,403.429,167.980,45.499,158.451
C03142=1027.894,37.769,403.446,167.977,45.501,158.451
C03143=1027.888,37.519,403.462,167.975,45.504,158.452
C03144=1027.882,37.270,403.479,167.972,45.506,158.452
C03145=1027.876,37.021,403.495,167.970,45.509,158.452
C03146=1027.870,36.771,403.511,167.967,45.511,158.452
C03147=1027.863,36.522,403.527,167.964,45.514,158.452
C03148=1027.857,36.273,403.543,167.962,45.516,158.452
C03149=1027.851,36.024,403.559,167.959,45.518,158.453
C03150=1027.844,35.774,403.575,167.957,45.521,158.453
C03151=1027.838,35.525,403.592,167.954,45.523,158.453
C03152=1027.833,35.275,403.607,167.952,45.526,158.453
C03153=1027.826,35.026,403.623,167.950,45.529,158.453
C03154=1027.820,34.776,403.639,167.947,45.531,158.454
C03155=1027.814,34.527,403.655,167.945,45.533,158.454
C03156=1027.807,34.278,403.671,167.942,45.535,158.454
C03157=1027.801,34.028,403.687,167.940,45.538,158.454
C03158=1027.795,33.779,403.703,167.938,45.541,158.454
C03159=1027.789,33.529,403.718,167.935,45.543,158.455
C03160=1027.782,33.279,403.735,167.933,45.545,158.455
C03161=1027.776,33.030,403.751,167.929,45.548,158.455
C03162=1027.770,32.781,403.767,167.927,45.550,158.455
C03163=1027.764,32.532,403.783,167.925,45.552,158.455
C03164=1027.758,32.282,403.799,167.922,45.555,158.456
C03165=1027.751,32.033,403.814,167.920,45.557,158.456
C03166=1027.746,31.783,403.831,167.917,45.560,158.456
C03167=1027.740,31.534,403.847,167.915,45.562,158.456
C03168=1027.733,31.285,403.863,167.913,45.564,158.456
C03169=1027.727,31.036,403.879,167.910,45.567,158.457
C03170=1027.721,30.786,403.894,167.908,45.569,158.457
C03171=1027.715,30.537,403.910,167.906,45.572,158.457
C03172=1027.709,30.287,403.926,167.903,45.574,158.457
C03173=1027.703,30.038,403.942,167.901,45.577,158.457
C03174=1027.696,29.788,403.957,167.898,45.579,158.457
C03175=1027.690,29.539,403.974,167.896,45.581,158.458
C03176=1027.684,29.290,403.990,167.893,45.583,158.458
C03177=1027.678,29.040,404.005,167.891,45.586,158.458
C03178=1027.672,28.791,404.021,167.887,45.588,158.458
C03179=1027.666,28.541,404.037,167.885,45.591,158.458
C03180=1027.659,28.292,404.053,167.883,45.593,158.458
C03181=1027.652,28.005,404.071,167.880,45.596,158.459
C03182=1027.646,27.720,404.089,167.877,45.599,158.459
C03183=1027.638,27.435,404.107,167.875,45.601,158.459
C03184=1027.631,27.149,404.125,167.871,45.604,158.459
C03185=1027.625,26.899,404.140,167.869,45.606,158.459
C03186=1027.619,26.650,404.156,167.867,45.609,158.460
C03187=1027.612,26.401,404.172,167.864,45.612,158.460
C03188=1027.607,26.151,404.188,167.862,45.614,158.460
C03189=1027.600,25.902,404.203,167.859,45.617,158.460
C03190=1027.594,25.652,404.219,167.857,45.619,158.460
C03191=1027.588,25.403,404.234,167.855,45.621,158.461
C03192=1027.582,25.153,404.250,167.851,45.624,158.461
C03193=1027.575,24.904,404.266,167.849,45.626,158.461
C03194=1027.569,24.654,404.281,167.846,45.629,158.461
C03195=1027.563,24.405,404.297,167.844,45.631,158.461
C03196=1027.556,24.155,404.312,167.842,45.634,158.462
C03197=1027.551,23.906,404.328,167.839,45.636,158.462
C03198=1027.544,23.656,404.343,167.837,45.638,158.462
C03199=1027.538,23.407,404.359,167.835,45.641,158.462
C03200=1027.532,23.158,404.374,167.832,45.643,158.462
C03201=1027.526,22.909,404.390,167.830,45.646,158.463
C03202=1027.520,22.659,404.405,167.826,45.648,158.463
C03203=1027.513,22.410,404.421,167.824,45.651,158.463
C03204=1027.508,22.160,404.436,167.821,45.653,158.463
C03205=1027.501,21.911,404.452,167.819,45.656,158.463
C03206=1027.495,21.661,404.467,167.816,45.658,158.463
C03207=1027.489,21.412,404.483,167.814,45.660,158.464
C03208=1027.482,21.162,404.498,167.812,45.662,158.464
C03209=1027.477,20.912,404.514,167.809,45.665,158.464
C03210=1027.470,20.663,404.529,167.807,45.667,158.464
C03211=1027.464,20.414,404.544,167.804,45.670,158.464
C03212=1027.458,20.165,404.560,167.801,45.672,158.464
C03213=1027.452,19.915,404.575,167.799,45.675,158.465
C03214=1027.446,19.665,404.591,167.796,45.678,158.465
C03215=1027.440,19.416,404.606,167.794,45.680,158.465
C03216=1027.433,19.167,404.621,167.792,45.682,158.465
C03217=1027.427,18.917,404.636,167.789,45.684,158.465
C03218=1027.421,18.668,404.652,167.787,45.687,158.466
C03219=1027.415,18.419,404.667,167.784,45.689,158.466
C03220=1027.409,18.169,404.682,167.781,45.692,158.466
C03221=1027.402,17.920,404.698,167.779,45.695,158.466
C03222=1027.396,17.670,404.713,167.776,45.697,158.466
C03223=1027.390,17.420,404.728,167.774,45.699,158.466
C03224=1027.384,17.171,404.743,167.771,45.701,158.467
C03225=1027.377,16.922,404.759,167.769,45.704,158.467
C03226=1027.372,16.672,404.774,167.766,45.706,158.467
C03227=1027.365,16.423,404.789,167.764,45.709,158.467
C03228=1027.359,16.173,404.804,167.761,45.711,158.467
C03229=1027.352,15.924,404.819,167.758,45.714,158.467
C03230=1027.347,15.674,404.835,167.756,45.717,158.468
C03231=1027.341,15.425,404.850,167.753,45.719,158.468
C03232=1027.335,15.175,404.865,167.751,45.721,158.468
C03233=1027.328,14.926,404.879,167.749,45.723,158.468
C03234=1027.322,14.676,404.896,167.746,45.726,158.468
C03235=1027.316,14.427,404.911,167.744,45.728,158.469
C03236=1027.310,14.178,404.925,167.740,45.731,158.469
C03237=1027.304,13.928,404.940,167.738,45.733,158.469
C03238=1027.298,13.678,404.956,167.736,45.736,158.469
C03239=1027.292,13.429,404.971,167.733,45.738,158.469
C03240=1027.285,13.179,404.986,167.731,45.741,158.469
C03241=1027.279,12.929,405.001,167.729,45.743,158.470
C03242=1027.273,12.681,405.016,167.725,45.746,158.470
C03243=1027.266,12.431,405.031,167.723,45.748,158.470
C03244=1027.260,12.182,405.046,167.720,45.751,158.470
C03245=1027.252,11.897,405.062,167.717,45.754,158.470
C03246=1027.246,11.612,405.079,167.715,45.757,158.471
C03247=1027.238,11.328,405.096,167.711,45.760,158.471
C03248=1027.232,11.044,405.113,167.709,45.762,158.471
C03249=1027.225,10.795,405.128,167.706,45.765,158.471
C03250=1027.219,10.545,405.143,167.703,45.767,158.471
C03251=1027.213,10.295,405.158,167.701,45.770,158.472
C03252=1027.207,10.046,405.172,167.699,45.773,158.472
C03253=1027.200,9.797,405.187,167.696,45.775,158.472
C03254=1027.194,9.547,405.202,167.693,45.778,158.472
C03255=1027.188,9.297,405.217,167.690,45.780,158.472
C03256=1027.182,9.048,405.232,167.688,45.783,158.473
C03257=1027.175,8.799,405.247,167.686,45.785,158.473
C03258=1027.168,8.549,405.261,167.683,45.787,158.473
C03259=1027.162,8.300,405.276,167.680,45.790,158.473
C03260=1027.156,8.051,405.290,167.678,45.793,158.473
C03261=1027.150,7.801,405.305,167.675,45.795,158.473
C03262=1027.144,7.551,405.320,167.673,45.798,158.474
C03263=1027.138,7.302,405.334,167.670,45.800,158.474
C03264=1027.132,7.052,405.349,167.668,45.803,158.474
C03265=1027.125,6.803,405.364,167.664,45.805,158.474
C03266=1027.119,6.554,405.379,167.662,45.808,158.474
C03267=1027.113,6.304,405.394,167.660,45.810,158.475
C03268=1027.107,6.054,405.409,167.657,45.812,158.475
C03269=1027.101,5.805,405.423,167.655,45.815,158.475
C03270=1027.095,5.555,405.437,167.652,45.817,158.475
C03271=1027.088,5.305,405.452,167.649,45.820,158.475
C03272=1027.083,5.056,405.467,167.647,45.823,158.475
C03273=1027.076,4.807,405.482,167.644,45.825,158.476
C03274=1027.070,4.557,405.497,167.642,45.828,158.476
C03275=1027.064,4.308,405.511,167.640,45.830,158.476
C03276=1027.058,4.058,405.526,167.636,45.833,158.476
C03277=1027.051,3.809,405.540,167.634,45.835,158.476
C03278=1027.045,3.560,405.554,167.632,45.837,158.476
C03279=1027.039,3.310,405.569,167.629,45.839,158.477
C03280=1027.033,3.061,405.584,167.627,45.842,158.477
C03281=1027.027,2.811,405.598,167.623,45.844,158.477
C03282=1027.020,2.561,405.613,167.621,45.847,158.477
C03283=1027.015,2.312,405.628,167.619,45.850,158.477
C03284=1027.008,2.062,405.643,167.616,45.852,158.477
C03285=1027.003,1.813,405.657,167.614,45.855,158.478
C03286=1026.996,1.563,405.672,167.611,45.857,158.478
C03287=1026.991,1.314,405.686,167.608,45.860,158.478
C03288=1026.985,1.064,405.700,167.605,45.862,158.478
C03289=1026.978,0.814,405.715,167.603,45.865,158.478
C03290=1026.972,0.565,405.730,167.601,45.867,158.478
C03291=1026.965,0.316,405.744,167.598,45.869,158.479
C03292=1026.960,0.066,405.758,167.595,45.872,158.479
C03293=1026.953,-0.183,405.773,167.592,45.874,158.479
C03294=1026.948,-0.432,405.788,167.590,45.876,158.479
C03295=1026.942,-0.682,405.802,167.588,45.879,158.479
C03296=1026.936,-0.931,405.816,167.585,45.881,158.479
C03297=1026.929,-1.181,405.831,167.583,45.883,158.479
C03298=1026.924,-1.431,405.845,167.579,45.886,158.480
C03299=1026.918,-1.680,405.860,167.577,45.888,158.480
C03300=1026.912,-1.929,405.875,167.574,45.891,158.480
C03301=1026.906,-2.179,405.889,167.572,45.893,158.480
C03302=1026.899,-2.428,405.903,167.570,45.896,158.480
C03303=1026.893,-2.678,405.917,167.567,45.898,158.480
C03304=1026.887,-2.927,405.932,167.564,45.901,158.481
C03305=1026.881,-3.177,405.947,167.561,45.903,158.481
C03306=1026.875,-3.427,405.961,167.559,45.906,158.481
C03307=1026.869,-3.676,405.976,167.556,45.908,158.481
C03308=1026.864,-3.926,405.989,167.554,45.910,158.481
C03309=1026.856,-4.208,406.006,167.551,45.913,158.481
C03310=1026.849,-4.491,406.022,167.547,45.916,158.481
C03311=1026.842,-4.774,406.037,167.545,45.918,158.482
C03312=1026.835,-5.056,406.054,167.542,45.921,158.482
C03313=1026.829,-5.305,406.067,167.539,45.924,158.482
C03314=1026.822,-5.555,406.082,167.536,45.927,158.482
C03315=1026.816,-5.804,406.095,167.534,45.929,158.482
C03316=1026.810,-6.054,406.110,167.531,45.932,158.483
C03317=1026.804,-6.303,406.124,167.529,45.935,158.483
C03318=1026.797,-6.553,406.138,167.525,45.937,158.483
C03319=1026.792,-6.802,406.152,167.523,45.940,158.483
C03320=1026.785,-7.052,406.166,167.521,45.942,158.483
C03321=1026.779,-7.302,406.180,167.517,45.945,158.483
C03322=1026.773,-7.550,406.194,167.515,45.947,158.484
C03323=1026.767,-7.800,406.208,167.513,45.949,158.484
C03324=1026.761,-8.050,406.221,167.510,45.952,158.484
C03325=1026.754,-8.299,406.236,167.507,45.955,158.484
C03326=1026.748,-8.549,406.250,167.504,45.957,158.484
C03327=1026.742,-8.799,406.264,167.502,45.960,158.485
C03328=1026.736,-9.048,406.278,167.500,45.962,158.485
C03329=1026.730,-9.297,406.292,167.496,45.965,158.485
C03330=1026.724,-9.547,406.306,167.494,45.968,158.485
C03331=1026.718,-9.797,406.319,167.491,45.970,158.485
C03332=1026.711,-10.046,406.334,167.489,45.973,158.485
C03333=1026.705,-10.296,406.347,167.486,45.975,158.485
C03334=1026.700,-10.545,406.361,167.483,45.978,158.486
C03335=1026.692,-10.795,406.376,167.481,45.980,158.486
C03336=1026.687,-11.044,406.390,167.478,45.983,158.486
C03337=1026.680,-11.294,406.403,167.475,45.985,158.486
C03338=1026.675,-11.544,406.417,167.473,45.987,158.486
C03339=1026.668,-11.792,406.431,167.470,45.990,158.487
C03340=1026.662,-12.043,406.445,167.467,45.992,158.487
C03341=1026.657,-12.292,406.459,167.465,45.995,158.487
C03342=1026.650,-12.541,406.472,167.462,45.997,158.487
C03343=1026.644,-12.792,406.487,167.460,46.000,158.487
C03344=1026.638,-13.040,406.501,167.457,46.003,158.487
C03345=1026.632,-13.290,406.514,167.454,46.005,158.487
C03346=1026.625,-13.540,406.528,167.452,46.008,158.488
C03347=1026.620,-13.789,406.542,167.449,46.010,158.488
C03348=1026.614,-14.039,406.555,167.446,46.013,158.488
C03349=1026.608,-14.289,406.569,167.443,46.015,158.488
C03350=1026.601,-14.538,406.583,167.441,46.018,158.488
C03351=1026.596,-14.787,406.597,167.437,46.020,158.488
C03352=1026.590,-15.036,406.611,167.435,46.023,158.488
C03353=1026.583,-15.287,406.625,167.433,46.025,158.489
C03354=1026.577,-15.536,406.638,167.430,46.027,158.489
C03355=1026.572,-15.786,406.652,167.427,46.030,158.489
C03356=1026.565,-16.036,406.666,167.425,46.033,158.489
C03357=1026.559,-16.285,406.679,167.422,46.035,158.489
C03358=1026.553,-16.534,406.693,167.419,46.038,158.489
C03359=1026.546,-16.784,406.706,167.416,46.040,158.490
C03360=1026.540,-17.034,406.720,167.414,46.043,158.490
C03361=1026.534,-17.283,406.733,167.411,46.045,158.490
C03362=1026.529,-17.532,406.747,167.408,46.048,158.490
C03363=1026.522,-17.782,406.760,167.406,46.051,158.490
C03364=1026.515,-18.032,406.774,167.403,46.053,158.490
C03365=1026.509,-18.281,406.787,167.400,46.056,158.491
C03366=1026.503,-18.531,406.801,167.398,46.059,158.491
C03367=1026.497,-18.781,406.814,167.394,46.061,158.491
C03368=1026.491,-19.030,406.828,167.392,46.064,158.491
C03369=1026.485,-19.280,406.840,167.390,46.066,158.491
C03370=1026.479,-19.530,406.854,167.386,46.069,158.491
C03371=1026.473,-19.779,406.868,167.384,46.072,158.492
C03372=1026.466,-20.028,406.881,167.382,46.074,158.492
C03373=1026.460,-20.309,406.896,167.378,46.077,158.492
C03374=1026.452,-20.590,406.912,167.375,46.080,158.492
C03375=1026.446,-20.871,406.927,167.372,46.083,158.492
C03376=1026.439,-21.151,406.941,167.369,46.085,158.492
C03377=1026.432,-21.401,406.955,167.366,46.088,158.493
C03378=1026.427,-21.650,406.968,167.364,46.091,158.493
C03379=1026.420,-21.900,406.982,167.361,46.093,158.493
C03380=1026.414,-22.150,406.995,167.358,46.096,158.493
C03381=1026.408,-22.399,407.008,167.355,46.098,158.493
C03382=1026.403,-22.649,407.022,167.353,46.101,158.493
C03383=1026.396,-22.898,407.035,167.350,46.103,158.493
C03384=1026.390,-23.148,407.048,167.347,46.106,158.494
C03385=1026.384,-23.398,407.061,167.345,46.109,158.494
C03386=1026.378,-23.648,407.075,167.341,46.111,158.494
C03387=1026.372,-23.897,407.088,167.339,46.114,158.494
C03388=1026.366,-24.146,407.102,167.337,46.116,158.494
C03389=1026.360,-24.395,407.115,167.333,46.119,158.494
C03390=1026.354,-24.645,407.127,167.331,46.122,158.495
C03391=1026.348,-24.895,407.141,167.329,46.124,158.495
C03392=1026.341,-25.145,407.155,167.325,46.127,158.495
C03393=1026.335,-25.395,407.168,167.323,46.129,158.495
C03394=1026.329,-25.644,407.181,167.320,46.132,158.495
C03395=1026.324,-25.894,407.195,167.317,46.134,158.495
C03396=1026.318,-26.143,407.208,167.315,46.137,158.496
C03397=1026.312,-26.393,407.220,167.312,46.139,158.496
C03398=1026.305,-26.642,407.234,167.309,46.142,158.496
C03399=1026.299,-26.891,407.247,167.306,46.144,158.496
C03400=1026.294,-27.141,407.260,167.304,46.147,158.496
C03401=1026.288,-27.391,407.273,167.301,46.150,158.496
C03402=1026.282,-27.640,407.287,167.298,46.152,158.496
C03403=1026.275,-27.891,407.300,167.295,46.155,158.497
C03404=1026.269,-28.140,407.313,167.293,46.157,158.497
C03405=1026.263,-28.390,407.325,167.290,46.159,158.497
C03406=1026.257,-28.639,407.339,167.287,46.162,158.497
C03407=1026.251,-28.889,407.351,167.285,46.165,158.497
C03408=1026.244,-29.138,407.364,167.281,46.167,158.497
C03409=1026.238,-29.388,407.377,167.279,46.170,158.498
C03410=1026.232,-29.637,407.390,167.276,46.173,158.498
C03411=1026.226,-29.887,407.402,167.273,46.176,158.498
C03412=1026.220,-30.136,407.416,167.271,46.178,158.498
C03413=1026.214,-30.386,407.428,167.267,46.181,158.498
C03414=1026.207,-30.635,407.441,167.265,46.184,158.498
C03415=1026.202,-30.885,407.454,167.263,46.186,158.499
C03416=1026.195,-31.134,407.467,167.259,46.189,158.499
C03417=1026.189,-31.384,407.480,167.257,46.192,158.499
C03418=1026.183,-31.634,407.493,167.253,46.194,158.499
C03419=1026.177,-31.883,407.506,167.251,46.197,158.499
C03420=1026.171,-32.133,407.519,167.249,46.200,158.499
C03421=1026.165,-32.383,407.531,167.245,46.202,158.499
C03422=1026.159,-32.633,407.544,167.243,46.205,158.500
C03423=1026.153,-32.882,407.557,167.240,46.207,158.500
C03424=1026.147,-33.132,407.570,167.237,46.210,158.500
C03425=1026.140,-33.381,407.583,167.234,46.213,158.500
C03426=1026.134,-33.630,407.595,167.231,46.215,158.500
C03427=1026.128,-33.880,407.608,167.229,46.218,158.500
C03428=1026.122,-34.130,407.621,167.226,46.221,158.501
C03429=1026.116,-34.380,407.633,167.223,46.223,158.501
C03430=1026.110,-34.629,407.647,167.220,46.226,158.501
C03431=1026.104,-34.879,407.659,167.218,46.228,158.501
C03432=1026.098,-35.129,407.672,167.215,46.230,158.501
C03433=1026.092,-35.378,407.685,167.212,46.233,158.501
C03434=1026.086,-35.628,407.698,167.209,46.236,158.501
C03435=1026.080,-35.878,407.710,167.206,46.239,158.502
C03436=1026.074,-36.127,407.723,167.204,46.241,158.502
C03437=1026.067,-36.407,407.737,167.200,46.244,158.502
C03438=1026.060,-36.687,407.751,167.197,46.247,158.502
C03439=1026.054,-36.967,407.765,167.195,46.249,158.502
C03440=1026.047,-37.247,407.780,167.191,46.252,158.502
C03441=1026.042,-37.496,407.792,167.188,46.255,158.502
C03442=1026.036,-37.746,407.805,167.186,46.258,158.503
C03443=1026.029,-37.995,407.818,167.182,46.261,158.503
C03444=1026.024,-38.245,407.830,167.180,46.263,158.503
C03445=1026.017,-38.494,407.842,167.178,46.265,158.503
C03446=1026.011,-38.744,407.855,167.174,46.268,158.503
C03447=1026.005,-38.994,407.868,167.172,46.271,158.503
C03448=1025.999,-39.243,407.881,167.168,46.274,158.503
C03449=1025.993,-39.493,407.893,167.166,46.276,158.504
C03450=1025.987,-39.742,407.905,167.163,46.279,158.504
C03451=1025.981,-39.992,407.917,167.160,46.281,158.504
C03452=1025.975,-40.242,407.930,167.157,46.284,158.504
C03453=1025.968,-40.492,407.942,167.155,46.287,158.504
C03454=1025.962,-40.741,407.954,167.152,46.289,158.504
C03455=1025.957,-40.991,407.967,167.149,46.292,158.505
C03456=1025.950,-41.241,407.979,167.147,46.295,158.505
C03457=1025.945,-41.490,407.991,167.143,46.298,158.505
C03458=1025.938,-41.739,408.004,167.141,46.300,158.505
C03459=1025.932,-41.989,408.016,167.138,46.303,158.505
C03460=1025.926,-42.239,408.029,167.135,46.306,158.505
C03461=1025.919,-42.488,408.041,167.132,46.308,158.505
C03462=1025.914,-42.738,408.053,167.130,46.311,158.506
C03463=1025.908,-42.987,408.066,167.126,46.314,158.506
C03464=1025.901,-43.237,408.078,167.124,46.317,158.506
C03465=1025.895,-43.487,408.090,167.120,46.319,158.506
C03466=1025.890,-43.737,408.103,167.118,46.322,158.506
C03467=1025.883,-43.986,408.114,167.115,46.325,158.506
C03468=1025.878,-44.236,408.127,167.112,46.327,158.507
C03469=1025.872,-44.485,408.139,167.109,46.330,158.507
C03470=1025.865,-44.735,408.151,167.107,46.333,158.507
C03471=1025.860,-44.985,408.163,167.103,46.335,158.507
C03472=1025.853,-45.234,408.175,167.101,46.338,158.507
C03473=1025.847,-45.484,408.187,167.098,46.341,158.507
C03474=1025.842,-45.734,408.200,167.095,46.343,158.507
C03475=1025.836,-45.983,408.212,167.092,46.346,158.508
C03476=1025.830,-46.233,408.224,167.090,46.349,158.508
C03477=1025.824,-46.483,408.237,167.086,46.351,158.508
C03478=1025.817,-46.732,408.249,167.084,46.354,158.508
C03479=1025.812,-46.982,408.261,167.082,46.357,158.508
C03480=1025.805,-47.231,408.273,167.078,46.359,158.508
C03481=1025.799,-47.481,408.285,167.076,46.362,158.509
C03482=1025.794,-47.731,408.297,167.072,46.365,158.509
C03483=1025.788,-47.980,408.309,167.070,46.367,158.509
C03484=1025.782,-48.230,408.321,167.067,46.370,158.509
C03485=1025.776,-48.479,408.333,167.064,46.373,158.509
C03486=1025.770,-48.729,408.345,167.061,46.375,158.509
C03487=1025.764,-48.979,408.358,167.059,46.378,158.509
C03488=1025.758,-49.228,408.369,167.055,46.380,158.509
C03489=1025.752,-49.478,408.381,167.053,46.383,158.510
C03490=1025.745,-49.728,408.393,167.049,46.386,158.510
C03491=1025.740,-49.977,408.406,167.047,46.388,158.510
C03492=1025.734,-50.227,408.418,167.044,46.391,158.510
C03493=1025.728,-50.477,408.429,167.041,46.394,158.510
C03494=1025.723,-50.726,408.442,167.038,46.396,158.510
C03495=1025.716,-50.976,408.454,167.036,46.399,158.510
C03496=1025.710,-51.226,408.465,167.032,46.402,158.511
C03497=1025.704,-51.475,408.477,167.030,46.405,158.511
C03498=1025.698,-51.725,408.488,167.027,46.408,158.511
C03499=1025.691,-51.975,408.500,167.023,46.411,158.511
C03500=1025.685,-52.224,408.512,167.021,46.413,158.511
C03501=1025.678,-52.505,408.524,167.018,46.417,158.512
C03502=1025.672,-52.785,408.538,167.015,46.420,158.512
C03503=1025.665,-53.066,408.551,167.011,46.423,158.512
C03504=1025.658,-53.346,408.564,167.008,46.426,158.512
C03505=1025.652,-53.596,408.575,167.005,46.429,158.512
C03506=1025.646,-53.845,408.587,167.001,46.432,158.512
C03507=1025.640,-54.095,408.599,166.999,46.435,158.513
C03508=1025.633,-54.345,408.611,166.996,46.438,158.513
C03509=1025.627,-54.594,408.622,166.994,46.441,158.513
C03510=1025.621,-54.844,408.634,166.990,46.443,158.513
C03511=1025.616,-55.093,408.646,166.988,46.446,158.513
C03512=1025.609,-55.343,408.657,166.985,46.449,158.513
C03513=1025.603,-55.593,408.669,166.981,46.452,158.513
C03514=1025.597,-55.842,408.680,166.979,46.454,158.514
C03515=1025.590,-56.092,408.691,166.976,46.458,158.514
C03516=1025.585,-56.342,408.703,166.973,46.460,158.514
C03517=1025.579,-56.592,408.714,166.970,46.463,158.514
C03518=1025.573,-56.841,408.726,166.967,46.466,158.514
C03519=1025.566,-57.091,408.737,166.964,46.468,158.514
C03520=1025.560,-57.340,408.749,166.961,46.472,158.515
C03521=1025.555,-57.590,408.761,166.959,46.474,158.515
C03522=1025.549,-57.839,408.772,166.955,46.477,158.515
C03523=1025.542,-58.089,408.784,166.952,46.480,158.515
C03524=1025.537,-58.339,408.794,166.950,46.482,158.515
C03525=1025.530,-58.588,408.806,166.947,46.486,158.515
C03526=1025.525,-58.838,408.818,166.944,46.488,158.516
C03527=1025.519,-59.088,408.829,166.941,46.491,158.516
C03528=1025.513,-59.337,408.841,166.937,46.494,158.516
C03529=1025.506,-59.587,408.852,166.935,46.496,158.516
C03530=1025.501,-59.837,408.863,166.932,46.500,158.516
C03531=1025.494,-60.086,408.875,166.930,46.502,158.516
C03532=1025.489,-60.336,408.886,166.926,46.505,158.516
C03533=1025.483,-60.586,408.897,166.924,46.507,158.517
C03534=1025.477,-60.835,408.909,166.921,46.511,158.517
C03535=1025.470,-61.085,408.920,166.917,46.514,158.517
C03536=1025.464,-61.335,408.931,166.915,46.516,158.517
C03537=1025.458,-61.585,408.943,166.911,46.519,158.517
C03538=1025.453,-61.834,408.955,166.909,46.521,158.517
C03539=1025.447,-62.084,408.966,166.906,46.525,158.517
C03540=1025.441,-62.334,408.977,166.903,46.528,158.518
C03541=1025.435,-62.583,408.988,166.900,46.530,158.518
C03542=1025.428,-62.833,409.000,166.897,46.533,158.518
C03543=1025.423,-63.083,409.010,166.895,46.536,158.518
C03544=1025.418,-63.332,409.022,166.891,46.539,158.518
C03545=1025.411,-63.582,409.034,166.888,46.541,158.518
C03546=1025.405,-63.831,409.045,166.885,46.544,158.518
C03547=1025.399,-64.082,409.056,166.882,46.547,158.519
C03548=1025.393,-64.331,409.067,166.880,46.550,158.519
C03549=1025.387,-64.581,409.078,166.876,46.552,158.519
C03550=1025.381,-64.831,409.090,166.874,46.555,158.519
C03551=1025.376,-65.080,409.101,166.871,46.558,158.519
C03552=1025.370,-65.329,409.112,166.868,46.561,158.519
C03553=1025.364,-65.580,409.123,166.865,46.563,158.519
C03554=1025.358,-65.829,409.134,166.862,46.566,158.520
C03555=1025.352,-66.079,409.145,166.860,46.569,158.520
C03556=1025.346,-66.328,409.157,166.856,46.572,158.520
C03557=1025.341,-66.578,409.169,166.853,46.574,158.520
C03558=1025.335,-66.828,409.179,166.850,46.577,158.520
C03559=1025.328,-67.078,409.191,166.847,46.580,158.520
C03560=1025.323,-67.327,409.202,166.845,46.582,158.520
C03561=1025.317,-67.577,409.212,166.841,46.585,158.520
C03562=1025.311,-67.826,409.223,166.839,46.588,158.521
C03563=1025.305,-68.076,409.235,166.836,46.591,158.521
C03564=1025.299,-68.326,409.245,166.832,46.593,158.521
C03565=1025.293,-68.607,409.259,166.829,46.596,158.521
C03566=1025.286,-68.889,409.271,166.826,46.599,158.521
C03567=1025.280,-69.171,409.283,166.822,46.602,158.521
C03568=1025.273,-69.451,409.296,166.819,46.606,158.522
C03569=1025.267,-69.701,409.307,166.817,46.608,158.522
C03570=1025.262,-69.951,409.319,166.814,46.611,158.522
C03571=1025.256,-70.201,409.329,166.810,46.614,158.522
C03572=1025.250,-70.450,409.340,166.808,46.617,158.522
C03573=1025.244,-70.700,409.352,166.805,46.620,158.522
C03574=1025.238,-70.950,409.362,166.802,46.622,158.522
C03575=1025.232,-71.199,409.373,166.799,46.625,158.522
C03576=1025.227,-71.449,409.384,166.796,46.628,158.523
C03577=1025.221,-71.698,409.395,166.793,46.631,158.523
C03578=1025.216,-71.949,409.406,166.790,46.633,158.523
C03579=1025.210,-72.199,409.417,166.787,46.636,158.523
C03580=1025.204,-72.448,409.428,166.784,46.639,158.523
C03581=1025.198,-72.698,409.439,166.782,46.641,158.523
C03582=1025.193,-72.947,409.450,166.778,46.644,158.523
C03583=1025.187,-73.197,409.461,166.776,46.647,158.524
C03584=1025.181,-73.447,409.472,166.772,46.649,158.523
C03585=1025.175,-73.697,409.483,166.769,46.652,158.524
C03586=1025.169,-73.946,409.494,166.767,46.655,158.524
C03587=1025.164,-74.196,409.505,166.763,46.657,158.524
C03588=1025.158,-74.446,409.515,166.761,46.660,158.524
C03589=1025.152,-74.695,409.525,166.758,46.663,158.524
C03590=1025.146,-74.945,409.537,166.755,46.666,158.524
C03591=1025.140,-75.195,409.548,166.752,46.669,158.525
C03592=1025.135,-75.445,409.558,166.749,46.672,158.525
C03593=1025.129,-75.694,409.569,166.746,46.675,158.525
C03594=1025.123,-75.944,409.579,166.743,46.677,158.525
C03595=1025.117,-76.194,409.589,166.740,46.680,158.525
C03596=1025.111,-76.443,409.600,166.737,46.684,158.525
C03597=1025.105,-76.693,409.611,166.734,46.686,158.525
C03598=1025.099,-76.943,409.622,166.731,46.689,158.526
C03599=1025.093,-77.193,409.632,166.728,46.692,158.526
C03600=1025.087,-77.442,409.642,166.725,46.695,158.526
C03601=1025.082,-77.692,409.653,166.722,46.698,158.526
C03602=1025.076,-77.942,409.664,166.719,46.701,158.526
C03603=1025.070,-78.191,409.674,166.717,46.703,158.526
C03604=1025.064,-78.441,409.684,166.713,46.707,158.526
C03605=1025.059,-78.690,409.695,166.710,46.709,158.526
C03606=1025.053,-78.940,409.706,166.708,46.712,158.527
C03607=1025.047,-79.190,409.716,166.704,46.715,158.527
C03608=1025.042,-79.440,409.727,166.701,46.718,158.527
C03609=1025.035,-79.689,409.737,166.699,46.721,158.527
C03610=1025.029,-79.940,409.748,166.695,46.724,158.527
C03611=1025.023,-80.189,409.758,166.692,46.726,158.527
C03612=1025.018,-80.439,409.769,166.690,46.729,158.527
C03613=1025.011,-80.688,409.779,166.686,46.732,158.528
C03614=1025.006,-80.938,409.789,166.683,46.735,158.528
C03615=1025.000,-81.188,409.799,166.680,46.738,158.528
C03616=1024.994,-81.438,409.809,166.678,46.741,158.528
C03617=1024.988,-81.688,409.819,166.674,46.744,158.528
C03618=1024.982,-81.937,409.830,166.671,46.747,158.528
C03619=1024.976,-82.187,409.840,166.668,46.750,158.528
C03620=1024.970,-82.436,409.850,166.666,46.753,158.529
C03621=1024.964,-82.686,409.860,166.662,46.756,158.529
C03622=1024.959,-82.936,409.870,166.659,46.759,158.529
C03623=1024.952,-83.185,409.880,166.657,46.762,158.529
C03624=1024.947,-83.436,409.891,166.653,46.765,158.529
C03625=1024.941,-83.685,409.901,166.650,46.768,158.529
C03626=1024.935,-83.935,409.911,166.647,46.771,158.530
C03627=1024.929,-84.185,409.921,166.645,46.774,158.530
C03628=1024.923,-84.434,409.931,166.641,46.777,158.530
C03629=1024.915,-84.787,409.945,166.637,46.781,158.530
C03630=1024.906,-85.139,409.960,166.632,46.785,158.530
C03631=1024.899,-85.491,409.974,166.629,46.790,158.531
C03632=1024.890,-85.842,409.988,166.625,46.794,158.531
C03633=1024.884,-86.093,409.998,166.621,46.797,158.531
C03634=1024.878,-86.342,410.008,166.618,46.800,158.531
C03635=1024.873,-86.592,410.019,166.616,46.803,158.531
C03636=1024.866,-86.842,410.028,166.612,46.806,158.532
C03637=1024.861,-87.092,410.038,166.609,46.809,158.532
